(* IEC 61131-3 sources: plc_simulator/services/codesys/POUs (part 4) *)

(* ---- STC_FC_DispatchTask.st ---- *)
(* ===========================================================================================
 *  STC_FC_DispatchTask — Validate and dispatch tasks to transporters
 *
 *  Company : Galvatek part of the John Cockerill Group
 *  Author  : Jarmo Piipponen
 *  Created : 25.03.2026
 *
 * -------------------------------------------------------------------------------------------
 *  Called every PLC scan from MainScheduler.
 *  For each idle transporter with queued tasks:
 *  1. Skip if transporter not idle or queue empty
 *  2. Time check: start_time close enough?
 *  3. Sink station free check (with parallel alternatives)
 *  4. Conflict check against active transporters
 *  5. Dispatch: write to TransporterStatus → RunTasks picks it up
 *
 *  ------------------------------------------------------------------------------------------
 *
 *  Changes:
 *
 *
 *
 *)

FUNCTION STC_FC_DispatchTask : BOOL

(* Introduction of Variables ----------------------------------------------------------------*)

VAR_EXTERNAL CONSTANT
    MAX_TRANSPORTERS        : INT;
    MAX_UNITS               : INT;
    MAX_STATIONS_PER_STEP   : INT;
    MAX_STEPS_PER_PROGRAM   : INT;
    MIN_STATION_INDEX        : INT;
    MAX_STATION_INDEX        : INT;
    SCH_DISPATCH_MARGIN_S   : REAL;
    USED                    : INT;
    PROCESSED               : INT;
END_VAR

VAR_EXTERNAL
  TransporterStatus             : ARRAY[1..MAX_TRANSPORTERS] OF UDT_TransporterStatusType;
  Task                    : ARRAY[1..MAX_TRANSPORTERS] OF UDT_JC_TskQueueType;
  Stations                 : ARRAY[MIN_STATION_INDEX..MAX_STATION_INDEX] OF UDT_StationType;
  StationOccupancy             : ARRAY[1..MAX_STATION_INDEX] OF UDT_JC_UnitAtStationType;
  Unit                    : ARRAY[1..MAX_UNITS] OF UDT_JC_UnitType;
  TreatmentPrograms                 : ARRAY[1..MAX_UNITS] OF UDT_TreatmentProgramType;
  Ntt                     : ARRAY[1..MAX_TRANSPORTERS] OF UDT_JC_NttTransporterType;
  Batch                   : ARRAY[1..MAX_UNITS] OF UDT_BatchType;
  Move                    : ARRAY[1..MAX_TRANSPORTERS] OF UDT_JC_MoveTimesType;
  Transporters                     : ARRAY[0..MAX_TRANSPORTERS] OF UDT_TransporterType;
  Schedule                : ARRAY[1..MAX_UNITS] OF UDT_JC_TskScheduleType;
  TimeS                  : LINT;
  EventPending           : UDT_JC_EventMsgType;
  EventPendingValid     : BOOL;
  DispatchedTask         : ARRAY[1..MAX_TRANSPORTERS] OF UDT_JC_DispatchedTaskType;
END_VAR

VAR
  vTi                        : INT;     (* transporter loop *)
  (* Task fields — read from queue[1] to avoid struct copy *)
  vTUnit                    : INT;
  vTStage                   : INT;
  vTLift                    : INT;
  vTSink                    : INT;
  vTStart                   : LINT;
  vTFinish                  : LINT;
  vTCalcTime               : DINT;
  (* Time check *)
  vTravelS                  : REAL;
  vMarginS                  : LINT;
  vFromIdx                  : INT;
  vToIdx                    : INT;
  (* Sink search *)
  vSinkStn                  : INT;
  vSinkFree                 : BOOL;
  vBestStn                  : INT;
  vBestChange               : LINT;
  vSi                        : INT;
  vCandStn                  : INT;
  vCandFree                 : BOOL;
  vUj                        : INT;
  vTgt                       : INT;
  vNttIdx                   : INT;     (* resolved NTT index (buffer 6/7/8) *)
  vNttCnt                   : INT;
  vNttFbCnt                : INT;
  (* Conflict check *)
  vConflict                  : BOOL;
  vCj                        : INT;
  vTaskMin                  : INT;     (* min station of our proposed task *)
  vTaskMax                  : INT;     (* max station of our proposed task *)
  (* Queue position loop *)
  vQi                        : INT;
  (* Shift-down after dispatch *)
  vSh                        : INT;
  (* Transfer time for batch progress bar *)
  vXferTotal                : REAL;
  (* Program stage number for event *)
  vProgStage                : INT;
  (* Manual task dispatch flag *)
  vUnitOk                   : BOOL;
END_VAR

FOR vTi := 1 TO MAX_TRANSPORTERS DO

  (* ── 1. Skip if not idle or queue empty ── *)
  (* Accept idle (Phase=0) OR move-away in progress (Phase=1, Status=3) *)
  IF (TransporterStatus[vTi].Phase = 0 OR (TransporterStatus[vTi].Phase = 1 AND TransporterStatus[vTi].Status = 3))
     AND Task[vTi].Count >= 1 THEN

    (* Try each queue position — skip blocked tasks, dispatch first feasible *)
    FOR vQi := 1 TO Task[vTi].Count DO

    (* Read task fields from queue position vQi *)
    vTUnit      := Task[vTi].Queue[vQi].Unit;
    vTStage     := Task[vTi].Queue[vQi].Stage;  (* schedule index *)
    vTLift      := Task[vTi].Queue[vQi].LiftStationTarget;
    vTSink      := Task[vTi].Queue[vQi].SinkStationTarget;
    vTStart     := Task[vTi].Queue[vQi].StartTime;
    vTFinish    := Task[vTi].Queue[vQi].FinishTime;
    vTCalcTime := Task[vTi].Queue[vQi].CalcTime;

    (* Queue[].Stage already contains ProgramStage (set by STC_FC_CreateTasks) *)
    vProgStage := vTStage;

    (* ── 1b. Lift station unit check — unit must be AT the lift station ── *)
    (* Manual tasks have Unit=0 → skip unit-location check *)
    (* NOTE: CODESYS does NOT short-circuit OR — use nested IFs *)
    vUnitOk := FALSE;
    IF vTUnit = 0 THEN
      vUnitOk := TRUE;
    ELSIF vTUnit >= 1 AND vTUnit <= MAX_UNITS THEN
      IF Unit[vTUnit].location = vTLift THEN
        vUnitOk := TRUE;
      END_IF;
    END_IF;

    IF vUnitOk THEN

    (* ── 2. Time check ── *)
    vTravelS := 0.0;
    IF TransporterStatus[vTi].CurrentStation > 0 AND vTLift > 0
       AND TransporterStatus[vTi].CurrentStation <> vTLift THEN
      vFromIdx := TransporterStatus[vTi].CurrentStation - MIN_STATION_INDEX;
      vToIdx   := vTLift - MIN_STATION_INDEX;
      IF vFromIdx >= 1 AND vFromIdx <= 30 AND vToIdx >= 1 AND vToIdx <= 30 THEN
        vTravelS := INT_TO_REAL(Move[vTi].Travel[vFromIdx].ToTime[vToIdx]) / 10.0;
      END_IF;
    END_IF;

    vMarginS := vTStart - TimeS;

    IF vMarginS <= REAL_TO_LINT(vTravelS + SCH_DISPATCH_MARGIN_S) THEN

      (* ── 3. Sink station free check ── *)
      vSinkStn := vTSink;
      vSinkFree := FALSE;

      IF vSinkStn >= MIN_STATION_INDEX AND vSinkStn <= MAX_STATION_INDEX THEN
        vSinkFree := TRUE;
        FOR vUj := 1 TO MAX_UNITS DO
          IF Unit[vUj].location = vSinkStn AND Unit[vUj].Status = USED THEN
            vSinkFree := FALSE;
          END_IF;
        END_FOR;
      END_IF;

      IF NOT vSinkFree THEN
        (* Search alternative parallel stations *)
        vBestStn := 0;
        vBestChange := LINT#2000000000;

        IF vProgStage >= 1 AND vProgStage <= MAX_STEPS_PER_PROGRAM
           AND vTUnit >= 1 AND vTUnit <= MAX_UNITS THEN
          (* Treatment task — look in TreatmentPrograms for parallel stations *)
          FOR vSi := 0 TO MAX_STATIONS_PER_STEP - 1 DO
            vCandStn := TreatmentPrograms[vTUnit].Steps[vProgStage].Stations[vSi];
            IF vCandStn > 0 AND vCandStn <> vTSink THEN
              IF vCandStn >= MIN_STATION_INDEX AND vCandStn <= MAX_STATION_INDEX THEN
                vCandFree := TRUE;
                FOR vUj := 1 TO MAX_UNITS DO
                  IF Unit[vUj].location = vCandStn AND Unit[vUj].Status = USED THEN
                    vCandFree := FALSE;
                  END_IF;
                END_FOR;
                IF vCandFree THEN
                  IF StationOccupancy[vCandStn].ChangeTime < vBestChange THEN
                    vBestChange := StationOccupancy[vCandStn].ChangeTime;
                    vBestStn := vCandStn;
                  END_IF;
                END_IF;
              END_IF;
            END_IF;
          END_FOR;

        ELSIF vProgStage = 0 AND vTUnit >= 1 AND vTUnit <= MAX_UNITS THEN
          (* No-treatment task — look in Ntt for alternatives *)
          vTgt := Unit[vTUnit].Target;
          IF vTgt >= 1 AND vTgt <= 5 THEN
            (* Resolve buffer NTT index like NoTreatment does *)
            IF vTgt = 2 THEN
              IF Batch[vTUnit].BatchCode = 0 THEN
                vNttIdx := 6;
              ELSIF Batch[vTUnit].State = PROCESSED THEN
                vNttIdx := 8;
              ELSE
                vNttIdx := 7;
              END_IF;
            ELSE
              vNttIdx := vTgt;
            END_IF;
            (* Check primary stations *)
            vNttCnt := Ntt[vTi].Target[vNttIdx].StationCount;
            FOR vSi := 1 TO vNttCnt DO
              IF vSi <= MAX_STATIONS_PER_STEP THEN
                vCandStn := Ntt[vTi].Target[vNttIdx].Stations[vSi];
                IF vCandStn > 0 AND vCandStn <> vTSink THEN
                  IF vCandStn >= MIN_STATION_INDEX AND vCandStn <= MAX_STATION_INDEX THEN
                    vCandFree := TRUE;
                    FOR vUj := 1 TO MAX_UNITS DO
                      IF Unit[vUj].location = vCandStn AND Unit[vUj].Status = USED THEN
                        vCandFree := FALSE;
                      END_IF;
                    END_FOR;
                    IF vCandFree THEN
                      IF StationOccupancy[vCandStn].ChangeTime < vBestChange THEN
                        vBestChange := StationOccupancy[vCandStn].ChangeTime;
                        vBestStn := vCandStn;
                      END_IF;
                    END_IF;
                  END_IF;
                END_IF;
              END_IF;
            END_FOR;
            (* Check fallback stations *)
            vNttFbCnt := Ntt[vTi].Target[vNttIdx].FallbackCount;
            FOR vSi := 1 TO vNttFbCnt DO
              IF vSi <= MAX_STATIONS_PER_STEP THEN
                vCandStn := Ntt[vTi].Target[vNttIdx].FallbackStations[vSi];
                IF vCandStn > 0 AND vCandStn <> vTSink THEN
                  IF vCandStn >= MIN_STATION_INDEX AND vCandStn <= MAX_STATION_INDEX THEN
                    vCandFree := TRUE;
                    FOR vUj := 1 TO MAX_UNITS DO
                      IF Unit[vUj].location = vCandStn AND Unit[vUj].Status = USED THEN
                        vCandFree := FALSE;
                      END_IF;
                    END_FOR;
                    IF vCandFree THEN
                      IF StationOccupancy[vCandStn].ChangeTime < vBestChange THEN
                        vBestChange := StationOccupancy[vCandStn].ChangeTime;
                        vBestStn := vCandStn;
                      END_IF;
                    END_IF;
                  END_IF;
                END_IF;
              END_IF;
            END_FOR;
          END_IF;
        END_IF;

        IF vBestStn > 0 THEN
          vSinkStn := vBestStn;
          vSinkFree := TRUE;
        END_IF;
      END_IF;  (* NOT vSinkFree *)

      IF vSinkFree THEN

        (* ── 4. Conflict check ── *)
        vConflict := FALSE;

        IF vTLift <= vSinkStn THEN
          vTaskMin := vTLift;
          vTaskMax := vSinkStn;
        ELSE
          vTaskMin := vSinkStn;
          vTaskMax := vTLift;
        END_IF;

        FOR vCj := 1 TO MAX_TRANSPORTERS DO
          IF vCj <> vTi AND TransporterStatus[vCj].Phase > 0 THEN

            (* a) T2's entire active task inside our range → vConflict *)
            IF TransporterStatus[vCj].LiftStationTarget >= vTaskMin
               AND TransporterStatus[vCj].LiftStationTarget <= vTaskMax
               AND TransporterStatus[vCj].SinkStationTarget >= vTaskMin
               AND TransporterStatus[vCj].SinkStationTarget <= vTaskMax THEN
              vConflict := TRUE;
            END_IF;

            (* b) T2 delivers to one of our exact stations → vConflict *)
            IF TransporterStatus[vCj].SinkStationTarget = vTLift
               OR TransporterStatus[vCj].SinkStationTarget = vSinkStn THEN
              vConflict := TRUE;
            END_IF;

          END_IF;
        END_FOR;

        IF NOT vConflict THEN
          (* ── 5. Dispatch: assign task to transporter ── *)
          TransporterStatus[vTi].TaskId      := vTStart;
          TransporterStatus[vTi].LiftStationTarget := vTLift;
          TransporterStatus[vTi].SinkStationTarget := vSinkStn;
          TransporterStatus[vTi].CurrentTaskFinishTime := Task[vTi].Queue[vQi].FinishTime;
          StationOccupancy[vTi].UnitId      := vTUnit;
          TransporterStatus[vTi].TaskRemainingTime := vTCalcTime;

          (* ── 5b. Fill dispatched task package ── *)
          DispatchedTask[vTi].TaskId           := vTStart;
          DispatchedTask[vTi].UnitId           := vTUnit;
          DispatchedTask[vTi].LiftStation      := vTLift;
          DispatchedTask[vTi].SinkStation      := vSinkStn;
          IF vTLift >= MIN_STATION_INDEX AND vTLift <= MAX_STATION_INDEX THEN
            DispatchedTask[vTi].LiftX              := Stations[vTLift].XPosition;
            DispatchedTask[vTi].LiftKind           := Stations[vTLift].DryWet;
            DispatchedTask[vTi].DroppingTime_x10   := Stations[vTLift].DrippingTime;
            DispatchedTask[vTi].LiftDeviceDelay_x10 := Stations[vTLift].DeviceDelay;
          END_IF;
          IF vSinkStn >= MIN_STATION_INDEX AND vSinkStn <= MAX_STATION_INDEX THEN
            DispatchedTask[vTi].SinkX              := Stations[vSinkStn].XPosition;
            DispatchedTask[vTi].SinkKind           := Stations[vSinkStn].DryWet;
            DispatchedTask[vTi].SinkDeviceDelay_x10 := Stations[vSinkStn].DeviceDelay;
          END_IF;
          DispatchedTask[vTi].DripTrayDelay_x10 := Transporters[vTi].DripTrayDelay;
          DispatchedTask[vTi].TreatmentTime    := vTCalcTime;
          DispatchedTask[vTi].MinTime          := Task[vTi].Queue[vQi].MinTime;
          DispatchedTask[vTi].MaxTime          := Task[vTi].Queue[vQi].MaxTime;
          DispatchedTask[vTi].NttPrimary       := Task[vTi].Queue[vQi].NttPrimary;
          IF vTUnit >= 1 AND vTUnit <= MAX_UNITS THEN
            DispatchedTask[vTi].BatchCode      := Batch[vTUnit].BatchCode;
            DispatchedTask[vTi].ProgramStage   := Batch[vTUnit].CurStage;
          ELSE
            DispatchedTask[vTi].BatchCode      := 0;
            DispatchedTask[vTi].ProgramStage   := 0;
          END_IF;
          DispatchedTask[vTi].Active           := TRUE;

          (* ── Emit TASK_DISPATCHED event (msg_type=1) ── *)
          vXferTotal := STC_FC_CalcTransferTime(
            iFromStn            := vTLift,
            iToStn              := vSinkStn,
            iMove                := Move[vTi],
            iFromDroppingX10   := Stations[vTLift].DrippingTime,
            iToDeviceDelayX10 := Stations[vSinkStn].DeviceDelay,
            iDripTrayDelayX10 := Transporters[vTi].DripTrayDelay
          );
          IF vXferTotal < 1.0 THEN
            vXferTotal := INT_TO_REAL(ABS(vSinkStn - vTLift)) * 8.0;
          END_IF;
  IF vXferTotal < 5.0 THEN vXferTotal := 60.0; END_IF;
          DispatchedTask[vTi].TransferTime_x10 := REAL_TO_DINT(vXferTotal * 10.0);
          IF NOT EventPendingValid THEN
            EventPending.MsgType := 1;
            EventPending.TsHi := LINT_TO_UINT(TimeS / LINT#65536);
            EventPending.TsLo := LINT_TO_UINT(TimeS MOD LINT#65536);
            EventPending.Payload[1]  := LINT_TO_INT(vTStart / LINT#65536);   (* TaskId_Hi *)
            EventPending.Payload[2]  := LINT_TO_INT(vTStart MOD LINT#65536);  (* TaskId_Lo *)
            EventPending.Payload[3]  := vTi;
            EventPending.Payload[4]  := vTUnit;
            EventPending.Payload[5]  := vTLift;
            EventPending.Payload[6]  := vSinkStn;
            IF vTUnit >= 1 AND vTUnit <= MAX_UNITS THEN
              vProgStage := Batch[vTUnit].CurStage;
              EventPending.Payload[7]  := vProgStage;
              EventPending.Payload[8]  := Batch[vTUnit].BatchCode;
            ELSE
              EventPending.Payload[7]  := 0;
              EventPending.Payload[8]  := 0;
            END_IF;
            EventPending.Payload[9]  := DINT_TO_INT(vTCalcTime);
            EventPending.Payload[10] := DINT_TO_INT(Task[vTi].Queue[vQi].MinTime);
            EventPending.Payload[11] := DINT_TO_INT(Task[vTi].Queue[vQi].MaxTime);
            EventPending.Payload[12] := REAL_TO_INT(vXferTotal);
            EventPendingValid := TRUE;
          END_IF;

          (* Copy station-specific timing from config *)
          IF vTLift >= MIN_STATION_INDEX AND vTLift <= MAX_STATION_INDEX THEN
            TransporterStatus[vTi].DrippingTime := Stations[vTLift].DrippingTime;
          END_IF;

          (* Shift queue: remove position vQi, move rest up *)
          FOR vSh := vQi + 1 TO Task[vTi].Count DO
            Task[vTi].Queue[vSh - 1] := Task[vTi].Queue[vSh];
          END_FOR;
          (* Clear last slot *)
          Task[vTi].Queue[Task[vTi].Count].Unit := 0;
          Task[vTi].Queue[Task[vTi].Count].Stage := 0;
          Task[vTi].Queue[Task[vTi].Count].SrcStage := 0;
          Task[vTi].Queue[Task[vTi].Count].LiftStationTarget := 0;
          Task[vTi].Queue[Task[vTi].Count].SinkStationTarget := 0;
          Task[vTi].Queue[Task[vTi].Count].StartTime := 0;
          Task[vTi].Queue[Task[vTi].Count].FinishTime := 0;
          Task[vTi].Queue[Task[vTi].Count].CalcTime := 0;
          Task[vTi].Queue[Task[vTi].Count].MinTime := 0;
          Task[vTi].Queue[Task[vTi].Count].MaxTime := 0;
          Task[vTi].Count := Task[vTi].Count - 1;
          EXIT;  (* dispatched — stop searching this queue *)

        END_IF;  (* NOT vConflict *)

      END_IF;  (* vSinkFree *)

    END_IF;  (* time check *)

    END_IF;  (* unit at lift station *)

    END_FOR;  (* vQi — try next queue position *)

  END_IF;  (* idle + queue *)

END_FOR;

STC_FC_DispatchTask := TRUE;

END_FUNCTION

(* ---- STC_FC_ManualTask.st ---- *)
(* ===========================================================================================
 *  STC_FC_ManualTask — Execute manual transport tasks from gateway
 *
 *  Company : Galvatek part of the John Cockerill Group
 *  Author  : Jarmo Piipponen
 *  Created : 25.03.2026
 *
 * -------------------------------------------------------------------------------------------
 *  For each transporter, checks ManualTask[vTi].Valid.
 *  If the transporter is idle (Phase=0), validates stations,
 *  calculates transfer time, and inserts a task into the queue
 *  (same pattern as TSK_FC_NoTreatment).
 *  Clears Valid after task is created, or on invalid input.
 *
 *  Called from TSK_FB_Scheduler phase 2200 (before NTT).
 *
 * ------------------------------------------------------------------------------------------
 *
 *  Changes:
 *
 *
 *
 *)

FUNCTION STC_FC_ManualTask : BOOL

(* Introduction of Variables ----------------------------------------------------------------*)

VAR_INPUT
  iTimeS                  : LINT;
END_VAR

VAR_IN_OUT
  ioTask                   : ARRAY[1..MAX_TRANSPORTERS] OF UDT_JC_TskQueueType;
END_VAR

VAR_EXTERNAL
  ManualTask             : ARRAY[1..MAX_TRANSPORTERS] OF UDT_JC_ManualTaskType;
  TransporterStatus             : ARRAY[1..MAX_TRANSPORTERS] OF UDT_TransporterStatusType;
  Move                    : ARRAY[1..MAX_TRANSPORTERS] OF UDT_JC_MoveTimesType;
  Unit                    : ARRAY[1..MAX_UNITS] OF UDT_JC_UnitType;
  Stations                  : ARRAY[MIN_STATION_INDEX..MAX_STATION_INDEX] OF UDT_StationType;
  Transporters              : ARRAY[0..MAX_TRANSPORTERS] OF UDT_TransporterType;
END_VAR

VAR_EXTERNAL CONSTANT
  MAX_TASK_QUEUE            : INT;
  MAX_UNITS                 : INT;
  USED                      : INT;
END_VAR

VAR
  vTi                        : INT;
  vAi                        : INT;
  vSh                        : INT;
  vLift                      : INT;
  vSink                      : INT;
  vCovers                    : BOOL;
  vTransPos                 : INT;
  vTmpMove                  : UDT_JC_MoveTimesType;
  vXferS                    : REAL;
  vTravelToLiftS          : REAL;
  vTaskStart                : LINT;
  vTaskEnd                  : LINT;
END_VAR

STC_FC_ManualTask := TRUE;

FOR vTi := 1 TO MAX_TRANSPORTERS DO
  IF NOT ManualTask[vTi].Valid THEN
    CONTINUE;
  END_IF;

  vLift := ManualTask[vTi].LiftStation;
  vSink := ManualTask[vTi].SinkStation;

  (* Validate station range *)
  IF vLift < MIN_STATION_INDEX OR vLift > MAX_STATION_INDEX
     OR vSink < MIN_STATION_INDEX OR vSink > MAX_STATION_INDEX
     OR vLift = vSink THEN
    ManualTask[vTi].Valid := FALSE;
    CONTINUE;
  END_IF;

  (* Transporter must be active and idle *)
  (* Transporter must be active and idle or in move-away *)
  IF NOT TransporterStatus[vTi].IsActive THEN
    CONTINUE;
  END_IF;
  IF TransporterStatus[vTi].Phase <> 0
     AND NOT (TransporterStatus[vTi].Phase = 1 AND TransporterStatus[vTi].Status = 3) THEN
    CONTINUE;  (* keep Valid — retry next cycle *)
  END_IF;

  (* Check vLift station is within transporter TaskArea *)
  vCovers := FALSE;
  FOR vAi := 1 TO 4 DO
    IF Transporters[vTi].TaskArea[vAi].MinLift > 0
       OR Transporters[vTi].TaskArea[vAi].MaxLift > 0 THEN
      IF vLift >= Transporters[vTi].TaskArea[vAi].MinLift
         AND vLift <= Transporters[vTi].TaskArea[vAi].MaxLift THEN
        vCovers := TRUE;
      END_IF;
    END_IF;
  END_FOR;

  IF NOT vCovers THEN
    ManualTask[vTi].Valid := FALSE;
    CONTINUE;
  END_IF;

  (* Calculate transfer time *)
  vTmpMove := Move[vTi];
  vXferS := STC_FC_CalcTransferTime(
    iFromStn            := vLift,
    iToStn              := vSink,
    iMove                := vTmpMove,
    iFromDroppingX10   := Stations[vLift].DrippingTime,
    iToDeviceDelayX10 := Stations[vSink].DeviceDelay,
    iDripTrayDelayX10 := Transporters[vTi].DripTrayDelay);

  (* Calculate travel-to-vLift: time for transporter to reach vLift station *)
  vTravelToLiftS := 0.0;
  vTransPos := TransporterStatus[vTi].CurrentStation;
  IF vTransPos > 0 AND vTransPos <> vLift THEN
    vTravelToLiftS := STC_FC_CalcHorizontalTravel(
      iFromStn := vTransPos,
      iToStn   := vLift,
      iMove     := vTmpMove);
  END_IF;

  vTaskStart := iTimeS + REAL_TO_LINT(vTravelToLiftS);
  vTaskEnd   := vTaskStart + REAL_TO_LINT(vXferS);

  (* Check vSink station is free — no unit occupying it *)
  vCovers := TRUE;  (* reuse variable as sink_free flag *)
  FOR vSh := 1 TO MAX_UNITS DO
    IF Unit[vSh].location = vSink AND Unit[vSh].Status = USED THEN
      vCovers := FALSE;
    END_IF;
  END_FOR;
  IF NOT vCovers THEN
    ManualTask[vTi].Valid := FALSE;
    CONTINUE;
  END_IF;

  (* Insert task at queue position 1 *)
  IF ioTask[vTi].Count < MAX_TASK_QUEUE THEN
    FOR vSh := ioTask[vTi].Count TO 1 BY -1 DO
      ioTask[vTi].Queue[vSh + 1] := ioTask[vTi].Queue[vSh];
    END_FOR;
    ioTask[vTi].Queue[1].Unit              := 0;
    ioTask[vTi].Queue[1].Stage             := 0;
    ioTask[vTi].Queue[1].LiftStationTarget := vLift;
    ioTask[vTi].Queue[1].SinkStationTarget := vSink;
    ioTask[vTi].Queue[1].StartTime         := vTaskStart;
    ioTask[vTi].Queue[1].FinishTime        := vTaskEnd;
    ioTask[vTi].Queue[1].CalcTime          := 0;
    ioTask[vTi].Queue[1].MinTime           := 0;
    ioTask[vTi].Queue[1].MaxTime           := 0;
    ioTask[vTi].Queue[1].NttPrimary        := 0;
    ioTask[vTi].Count := ioTask[vTi].Count + 1;
  END_IF;

  ManualTask[vTi].Valid := FALSE;
END_FOR;

END_FUNCTION

(* ---- STC_FC_NoTreatmentStates.st ---- *)
(* ===========================================================================================
 *  STC_FC_NoTreatmentStates — Non-treatment target state management
 *
 *  Company : Galvatek part of the John Cockerill Group
 *  Author  : Jarmo Piipponen
 *  Created : 25.03.2026
 *
 * -------------------------------------------------------------------------------------------
 *  Manages non-treatment target states for all units.
 *
 *  Structure:
 *  Pass 0 — SNAPSHOT: read unit/batch/station state into vSnap[]
 *  Section 1 — PROCESSED: mark last-stage units as PROCESSED
 *  Section 2 — TO_AVOID: clear occupied next-stage stations
 *  Section 3 — TO_LOADING: route one empty unit to loading
 *
 *  ------------------------------------------------------------------------------------------
 *
 *  Changes:
 *
 *
 *
 *)

FUNCTION STC_FC_NoTreatmentStates : BOOL

(* Introduction of Variables ----------------------------------------------------------------*)

VAR_EXTERNAL CONSTANT
    MAX_UNITS               : INT;
    MAX_STEPS_PER_PROGRAM   : INT;
    MAX_STATIONS_PER_STEP   : INT;
    MIN_STATION_INDEX        : INT;
    MAX_STATION_INDEX        : INT;
    IN_PROCESS              : INT;
    PROCESSED               : INT;
    NOT_USED                : INT;
    TO_NONE                 : INT;
    TO_UNLOAD               : INT;
    TO_AVOID                : INT;
    TO_LOADING              : INT;
    USED                    : INT;
    OP_BUFFER               : INT;
    OP_BUFFER_PROCESSED     : INT;
    OP_LOADING              : INT;
    OP_LOADING_UNLOADING    : INT;
END_VAR

VAR_EXTERNAL
  Unit                    : ARRAY[1..MAX_UNITS] OF UDT_JC_UnitType;
  Batch                   : ARRAY[1..MAX_UNITS] OF UDT_BatchType;
  TreatmentPrograms                 : ARRAY[1..MAX_UNITS] OF UDT_TreatmentProgramType;
  Stations                 : ARRAY[MIN_STATION_INDEX..MAX_STATION_INDEX] OF UDT_StationType;
  StationOccupancy             : ARRAY[1..MAX_STATION_INDEX] OF UDT_JC_UnitAtStationType;
  TimeS                  : LINT;
  ProductionQueue        : INT;
  EventPending           : UDT_JC_EventMsgType;
  EventPendingValid     : BOOL;
END_VAR

VAR
  (* Snapshot *)
  vSnap                      : ARRAY[1..MAX_UNITS] OF UDT_JC_UnitSnapType;
  vU                         : INT;        (* unit loop index *)
  vHasLoading               : BOOL;       (* any unit already has TO_LOADING *)
  (* Section 1+2 *)
  vP                         : INT;        (* parallel station loop *)
  vNextStn                  : INT;        (* next stage station *)
  vOccUid                   : INT;        (* unit_id at an occupied station *)
  vFreeFound                : BOOL;       (* any next-stage station is free *)
  vAvoidUid                 : INT;        (* unit to mark TO_AVOID *)
  (* Section 3 *)
  vLoadFree                 : BOOL;       (* a loading station is free *)
  vLoadUid                  : INT;        (* best candidate for TO_LOADING *)
  vLoadInBuf               : BOOL;       (* current candidate is in buffer *)
  vStk                       : INT;        (* station loop *)
  vOp                        : INT;        (* station operation code *)
END_VAR

  (* ════════════════════════════════════════════════════════════
     Pass 0 — SNAPSHOT: collect per-unit state in one pass
     ════════════════════════════════════════════════════════════ *)
  vHasLoading := FALSE;

  FOR vU := 1 TO MAX_UNITS DO
    vSnap[vU].IsActive := Unit[vU].Status <> NOT_USED;
    IF NOT vSnap[vU].IsActive THEN
      CONTINUE;
    END_IF;

    vSnap[vU].Location       := Unit[vU].location;
    vSnap[vU].Target       := Unit[vU].Target;
    vSnap[vU].HasBatch := Batch[vU].BatchCode <> 0;
    vSnap[vU].BatchState    := Batch[vU].State;
    vSnap[vU].CurStage := Batch[vU].CurStage;

    vSnap[vU].OnStation := vSnap[vU].Location >= MIN_STATION_INDEX
                          AND vSnap[vU].Location <= MAX_STATION_INDEX;
    IF vSnap[vU].OnStation THEN
      vSnap[vU].LocationOp    := Stations[vSnap[vU].Location].StationType;
      vSnap[vU].InBuffer := vSnap[vU].LocationOp >= OP_BUFFER AND vSnap[vU].LocationOp <= OP_BUFFER_PROCESSED;
      IF StationOccupancy[vSnap[vU].Location].ChangeTime > 0 THEN
        vSnap[vU].Elapsed := TimeS - StationOccupancy[vSnap[vU].Location].ChangeTime;
      ELSE
        vSnap[vU].Elapsed := 0;
      END_IF;
      IF vSnap[vU].CurStage >= 1 THEN
        vSnap[vU].CalTime := TreatmentPrograms[vU].Steps[vSnap[vU].CurStage].CalTime;
      ELSE
        vSnap[vU].CalTime := 0;
      END_IF;
    ELSE
      vSnap[vU].LocationOp    := 0;
      vSnap[vU].InBuffer := FALSE;
      vSnap[vU].Elapsed   := 0;
      vSnap[vU].CalTime       := 0;
    END_IF;

    IF vSnap[vU].Target = TO_LOADING THEN
      vHasLoading := TRUE;
    END_IF;
  END_FOR;

  (* ════════════════════════════════════════════════════════════
     Section 1 — PROCESSED: mark batch done at last treatment stage
     ════════════════════════════════════════════════════════════ *)
  FOR vU := 1 TO MAX_UNITS DO
    IF NOT vSnap[vU].IsActive OR NOT vSnap[vU].HasBatch THEN
      CONTINUE;
    END_IF;
    IF vSnap[vU].BatchState <> IN_PROCESS OR NOT vSnap[vU].OnStation THEN
      CONTINUE;
    END_IF;
    IF vSnap[vU].CurStage >= 1 AND vSnap[vU].CurStage < MAX_STEPS_PER_PROGRAM THEN
      IF vSnap[vU].CurStage >= TreatmentPrograms[vU].StepCount THEN
        IF vSnap[vU].Elapsed > 0 AND vSnap[vU].Elapsed >= DINT_TO_LINT(vSnap[vU].CalTime) THEN
          Batch[vU].State := PROCESSED;
          vSnap[vU].BatchState   := PROCESSED;  (* update snapshot *)

          (* ── Emit BATCH_COMPLETED event (msg_type=5) ── *)
          IF NOT EventPendingValid THEN
            EventPending.MsgType := 5;
            EventPending.TsHi := LINT_TO_UINT(TimeS / LINT#65536);
            EventPending.TsLo := LINT_TO_UINT(TimeS MOD LINT#65536);
            EventPending.Payload[1]  := vU;                                  (* unit_id *)
            EventPending.Payload[2]  := Batch[vU].BatchCode;               (* batch_code *)
            EventPending.Payload[3]  := TreatmentPrograms[vU].StepCount;             (* stage_count *)
            EventPending.Payload[4]  := vSnap[vU].Location;                   (* final_station *)
            EventPending.Payload[5]  := 0;
            EventPending.Payload[6]  := 0;
            EventPending.Payload[7]  := 0;
            EventPending.Payload[8]  := 0;
            EventPending.Payload[9]  := 0;
            EventPending.Payload[10] := 0;
            EventPending.Payload[11] := 0;
            EventPending.Payload[12] := 0;
            EventPendingValid := TRUE;
          END_IF;

          (* Route to unloading station *)
          IF vSnap[vU].Target = TO_NONE THEN
            Unit[vU].Target := TO_UNLOAD;
            vSnap[vU].Target   := TO_UNLOAD;
          END_IF;
        END_IF;
      END_IF;
    END_IF;
  END_FOR;

  (* ════════════════════════════════════════════════════════════
     Section 2 — TO_AVOID: clear the way to next treatment station
     ════════════════════════════════════════════════════════════ *)
  FOR vU := 1 TO MAX_UNITS DO
    IF NOT vSnap[vU].IsActive OR NOT vSnap[vU].HasBatch THEN
      CONTINUE;
    END_IF;
    IF vSnap[vU].BatchState <> IN_PROCESS THEN
      CONTINUE;
    END_IF;
    IF vSnap[vU].CurStage < 1 OR vSnap[vU].CurStage >= MAX_STEPS_PER_PROGRAM THEN
      CONTINUE;
    END_IF;
    IF vSnap[vU].CurStage >= TreatmentPrograms[vU].StepCount THEN
      CONTINUE;  (* no next stage *)
    END_IF;

    (* — Pass 1: any next-stage station free or being cleared? — *)
    vFreeFound := FALSE;
    vAvoidUid  := 0;
    FOR vP := 0 TO MAX_STATIONS_PER_STEP - 1 DO
      vNextStn := TreatmentPrograms[vU].Steps[vSnap[vU].CurStage + 1].Stations[vP];
      IF vNextStn = 0 THEN
        EXIT;
      END_IF;
      IF vNextStn >= MIN_STATION_INDEX AND vNextStn <= MAX_STATION_INDEX THEN
        IF StationOccupancy[vNextStn].UnitId = 0 THEN
          vFreeFound := TRUE;
          EXIT;
        END_IF;
        vOccUid := StationOccupancy[vNextStn].UnitId;
        IF vOccUid >= 1 AND vOccUid <= MAX_UNITS THEN
          IF vSnap[vOccUid].Target = TO_AVOID THEN
            vFreeFound := TRUE;
            EXIT;
          END_IF;
        END_IF;
      END_IF;
    END_FOR;

    (* — Pass 2: all occupied → mark ONE movable unit TO_AVOID — *)
    IF NOT vFreeFound THEN
      FOR vP := 0 TO MAX_STATIONS_PER_STEP - 1 DO
        vNextStn := TreatmentPrograms[vU].Steps[vSnap[vU].CurStage + 1].Stations[vP];
        IF vNextStn = 0 THEN
          EXIT;
        END_IF;
        IF vNextStn >= MIN_STATION_INDEX AND vNextStn <= MAX_STATION_INDEX THEN
          vOccUid := StationOccupancy[vNextStn].UnitId;
          IF vOccUid >= 1 AND vOccUid <= MAX_UNITS THEN
            IF NOT vSnap[vOccUid].HasBatch AND vSnap[vOccUid].Target = TO_NONE THEN
              vAvoidUid := vOccUid;
              EXIT;
            END_IF;
          END_IF;
        END_IF;
      END_FOR;

      IF vAvoidUid >= 1 THEN
        Unit[vAvoidUid].Target := TO_AVOID;
        vSnap[vAvoidUid].Target     := TO_AVOID;  (* update snapshot *)
      END_IF;
    END_IF;
  END_FOR;

  (* ════════════════════════════════════════════════════════════
     Section 3 — TO_LOADING: route one empty unit to loading station
     ════════════════════════════════════════════════════════════ *)
  IF ProductionQueue = 1 AND NOT vHasLoading THEN

    (* Check if any loading station is free *)
    vLoadFree := FALSE;
    FOR vStk := MIN_STATION_INDEX TO MAX_STATION_INDEX DO
      vOp := Stations[vStk].StationType;
      IF (vOp = OP_LOADING OR vOp = OP_LOADING_UNLOADING)
         AND StationOccupancy[vStk].UnitId = 0 THEN
        vLoadFree := TRUE;
        EXIT;
      END_IF;
    END_FOR;

    IF vLoadFree THEN
      vLoadUid    := 0;
      vLoadInBuf := FALSE;
      FOR vU := 1 TO MAX_UNITS DO
        IF vSnap[vU].IsActive AND NOT vSnap[vU].HasBatch
           AND vSnap[vU].Target = TO_NONE AND vSnap[vU].OnStation THEN
          IF vSnap[vU].InBuffer THEN
            IF vLoadUid = 0 THEN
              vLoadUid    := vU;
              vLoadInBuf := TRUE;
            END_IF;
          ELSE
            IF vLoadUid = 0 OR vLoadInBuf THEN
              vLoadUid    := vU;
              vLoadInBuf := FALSE;
            END_IF;
          END_IF;
        END_IF;
      END_FOR;

      IF vLoadUid >= 1 THEN
        Unit[vLoadUid].Target := TO_LOADING;
      END_IF;
    END_IF; (* vLoadFree *)

  END_IF; (* production_queue AND NOT vHasLoading *)

  STC_FC_NoTreatmentStates := TRUE;

END_FUNCTION

(* ---- STC_FC_ShiftSchedule.st ---- *)
(* ===========================================================================================
 *  STC_FC_ShiftSchedule — Shift schedule + task times
 *
 *  Company : Galvatek part of the John Cockerill Group
 *  Author  : Jarmo Piipponen
 *  Created : 25.03.2026
 *
 * -------------------------------------------------------------------------------------------
 *  Propagates a time shift through one unit's schedule stages
 *  AND through all matching tasks.
 *
 *  Positive iAmount = DELAY (shift later),
 *  Negative iAmount = ADVANCE (shift earlier).
 *
 *  VAR_IN_OUT: ioSchedule, ioTask — caller passes live or
 *  workspace arrays.
 *
 *  ------------------------------------------------------------------------------------------
 *
 *  Changes:
 *
 *
 *
 *)

FUNCTION STC_FC_ShiftSchedule : BOOL

(* Introduction of Variables ----------------------------------------------------------------*)

VAR_INPUT
  iUnit                    : INT;     (* unit index 1..10 *)
  iFromStage              : INT;     (* propagate from this stage onward *)
  iAmount                  : REAL;    (* seconds to shift (+ = later, - = earlier) *)
END_VAR

VAR_IN_OUT  (* array sizes must match GVL_JC_Constants: 10=MAX_UNITS, 3=MAX_TRANSPORTERS *)
  ioSchedule               : ARRAY[1..10] OF UDT_JC_TskScheduleType;
  ioTask                   : ARRAY[1..3] OF UDT_JC_TskQueueType;
END_VAR

VAR_EXTERNAL CONSTANT
    MAX_TRANSPORTERS        : INT;
    MAX_UNITS               : INT;
END_VAR

VAR_EXTERNAL
  TimeS                  : LINT;
END_VAR

VAR
  vSc                        : INT;
  vSi                        : INT;
  vQi                        : INT;
  vTi                        : INT;
  vDuration                  : LINT;
END_VAR

STC_FC_ShiftSchedule := TRUE;
IF iUnit < 1 OR iUnit > MAX_UNITS THEN RETURN; END_IF;
IF ABS(iAmount) < 0.001 THEN RETURN; END_IF;

(* -- Shift schedule stages entry/exit times -- *)
vSc := ioSchedule[iUnit].StageCount;
FOR vSi := 1 TO vSc DO
  IF vSi >= 1 AND vSi <= 30
     AND ioSchedule[iUnit].Stages[vSi].ProgramStage >= iFromStage THEN
    ioSchedule[iUnit].Stages[vSi].EntryTime :=
      ioSchedule[iUnit].Stages[vSi].EntryTime + REAL_TO_LINT(iAmount);
    ioSchedule[iUnit].Stages[vSi].ExitTime :=
      ioSchedule[iUnit].Stages[vSi].ExitTime + REAL_TO_LINT(iAmount);
    (* GAP-3: Past-clamp -- don't let EntryTime go before now+1 *)
    IF iAmount < 0.0 AND ioSchedule[iUnit].Stages[vSi].EntryTime < TimeS + LINT#1 THEN
      ioSchedule[iUnit].Stages[vSi].ExitTime := TimeS + LINT#1
        + (ioSchedule[iUnit].Stages[vSi].ExitTime - ioSchedule[iUnit].Stages[vSi].EntryTime);
      ioSchedule[iUnit].Stages[vSi].EntryTime := TimeS + LINT#1;
    END_IF;
  END_IF;
END_FOR;

(* -- Shift matching tasks in all transporter queues -- *)
FOR vTi := 1 TO MAX_TRANSPORTERS DO
  FOR vQi := 1 TO ioTask[vTi].Count DO
    IF ioTask[vTi].Queue[vQi].Unit = iUnit
       AND ioTask[vTi].Queue[vQi].Stage >= iFromStage THEN
      ioTask[vTi].Queue[vQi].StartTime :=
        ioTask[vTi].Queue[vQi].StartTime + REAL_TO_LINT(iAmount);
      ioTask[vTi].Queue[vQi].FinishTime :=
        ioTask[vTi].Queue[vQi].FinishTime + REAL_TO_LINT(iAmount);
      (* GAP-3: Past-clamp -- don't let StartTime go before now+1 *)
      IF iAmount < 0.0 AND ioTask[vTi].Queue[vQi].StartTime < TimeS + LINT#1 THEN
        vDuration := ioTask[vTi].Queue[vQi].FinishTime - ioTask[vTi].Queue[vQi].StartTime;
        ioTask[vTi].Queue[vQi].StartTime := TimeS + LINT#1;
        ioTask[vTi].Queue[vQi].FinishTime := TimeS + LINT#1 + vDuration;
      END_IF;
    END_IF;
  END_FOR;
END_FOR;

END_FUNCTION

(* ---- STC_FC_SortTasks.st ---- *)
(* ===========================================================================================
 *  STC_FC_SortTasks — Insertion sort task queues by priority
 *
 *  Company : Galvatek part of the John Cockerill Group
 *  Author  : Jarmo Piipponen
 *  Created : 25.03.2026
 *
 * -------------------------------------------------------------------------------------------
 *  Shared FC: both TSK and DEP call this with different arrays.
 *  Priority: emergency (overtime ratio > 1.0) first, then
 *  earliest StartTime.
 *
 *  ------------------------------------------------------------------------------------------
 *
 *  Changes:
 *
 *
 *
 *)

FUNCTION STC_FC_SortTasks : BOOL

(* Introduction of Variables ----------------------------------------------------------------*)

VAR_INPUT
  iTrans                   : INT;    (* 0 = all, 1..3 = specific transporter *)
  iTimeS                  : LINT;
END_VAR

VAR_IN_OUT  (* array sizes must match GVL_JC_Constants: 3=MAX_TRANSPORTERS, 10=MAX_UNITS *)
  ioTask                   : ARRAY[1..3] OF UDT_JC_TskQueueType;
  ioBatch                  : ARRAY[1..10] OF UDT_BatchType;
END_VAR

VAR_EXTERNAL CONSTANT
    MAX_TRANSPORTERS        : INT;
    MAX_UNITS               : INT;
    IN_PROCESS              : INT;
END_VAR

VAR_EXTERNAL
  Unit                    : ARRAY[1..MAX_UNITS] OF UDT_JC_UnitType;
END_VAR

VAR
  vTi                        : INT;
  vTStart                   : INT;
  vTEnd                     : INT;
  vInsI                     : INT;
  vInsJ                     : INT;
  vInsCnt                   : INT;
  vTmpTask                  : UDT_JC_TskTaskType;
  vTmpUnit                  : INT;
  vCurUnit                  : INT;
  vTmpRatio                 : REAL;
  vCurRatio                 : REAL;
  vTmpEmerg                 : BOOL;
  vCurEmerg                 : BOOL;
  vDoShift                  : BOOL;
END_VAR

STC_FC_SortTasks := TRUE;

IF iTrans >= 1 AND iTrans <= 3 THEN
  vTStart := iTrans;
  vTEnd   := iTrans;
ELSE
  vTStart := 1;
  vTEnd   := 3;
END_IF;

FOR vTi := vTStart TO vTEnd DO
  vInsCnt := ioTask[vTi].Count;
  IF vInsCnt >= 2 THEN
    FOR vInsI := 2 TO vInsCnt DO
      vTmpTask := ioTask[vTi].Queue[vInsI];

      vTmpRatio := 0.0;
      vTmpUnit  := vTmpTask.Unit;
      IF vTmpUnit >= 1 AND vTmpUnit <= MAX_UNITS THEN
        IF ioBatch[vTmpUnit].State = IN_PROCESS
           AND vTmpTask.Stage >= 1 THEN
          IF ioBatch[vTmpUnit].CurStage = vTmpTask.Stage
             AND Unit[vTmpUnit].location = vTmpTask.LiftStationTarget
             AND ioBatch[vTmpUnit].StartTime > LINT#0
             AND ioBatch[vTmpUnit].MaxTime > 0 THEN
            vTmpRatio := LINT_TO_REAL(iTimeS - ioBatch[vTmpUnit].StartTime)
                         / DINT_TO_REAL(ioBatch[vTmpUnit].MaxTime);
          END_IF;
        END_IF;
      END_IF;
      vTmpEmerg := vTmpRatio > 1.0;

      vInsJ := 0;
      FOR vInsJ := vInsI - 1 TO 1 BY -1 DO
        vCurRatio := 0.0;
        vCurUnit  := ioTask[vTi].Queue[vInsJ].Unit;
        IF vCurUnit >= 1 AND vCurUnit <= MAX_UNITS THEN
          IF ioBatch[vCurUnit].State = IN_PROCESS
             AND ioTask[vTi].Queue[vInsJ].Stage >= 1 THEN
            IF ioBatch[vCurUnit].CurStage = ioTask[vTi].Queue[vInsJ].Stage
               AND Unit[vCurUnit].location = ioTask[vTi].Queue[vInsJ].LiftStationTarget
               AND ioBatch[vCurUnit].StartTime > LINT#0
               AND ioBatch[vCurUnit].MaxTime > 0 THEN
              vCurRatio := LINT_TO_REAL(iTimeS - ioBatch[vCurUnit].StartTime)
                           / DINT_TO_REAL(ioBatch[vCurUnit].MaxTime);
            END_IF;
          END_IF;
        END_IF;
        vCurEmerg := vCurRatio > 1.0;

        vDoShift := FALSE;
        IF vTmpEmerg AND NOT vCurEmerg THEN
          vDoShift := TRUE;
        ELSIF vTmpEmerg AND vCurEmerg THEN
          IF vTmpRatio > vCurRatio THEN
            vDoShift := TRUE;
          END_IF;
        ELSIF NOT vTmpEmerg AND NOT vCurEmerg THEN
          IF ioTask[vTi].Queue[vInsJ].StartTime > vTmpTask.StartTime THEN
            vDoShift := TRUE;
          END_IF;
        END_IF;

        IF NOT vDoShift THEN EXIT; END_IF;

        ioTask[vTi].Queue[vInsJ + 1] := ioTask[vTi].Queue[vInsJ];
      END_FOR;

      ioTask[vTi].Queue[vInsJ + 1] := vTmpTask;
    END_FOR;
  END_IF;
END_FOR;

END_FUNCTION

(* ---- STC_FC_SwapTasks.st ---- *)
(* ===========================================================================================
 *  STC_FC_SwapTasks — Swap same-station task pairs
 *
 *  Company : Galvatek part of the John Cockerill Group
 *  Author  : Jarmo Piipponen
 *  Created : 25.03.2026
 *
 * -------------------------------------------------------------------------------------------
 *  Shared FC: both TSK and DEP call this with different arrays.
 *  Swaps adjacent tasks on the same transporter when the first
 *  task's sink equals the second task's lift (chain optimization).
 *  Returns swap count.
 *
 *  ------------------------------------------------------------------------------------------
 *
 *  Changes:
 *
 *
 *
 *)

FUNCTION STC_FC_SwapTasks : INT   (* returns swap count *)

(* Introduction of Variables ----------------------------------------------------------------*)

VAR_IN_OUT  (* array sizes must match GVL_JC_Constants: 3=MAX_TRANSPORTERS *)
  ioTask                   : ARRAY[1..3] OF UDT_JC_TskQueueType;
END_VAR

VAR_EXTERNAL CONSTANT
    MAX_TRANSPORTERS        : INT;
END_VAR

VAR
  vTi                        : INT;
  vQi                        : INT;
  vCnt                       : INT;
  vTmp                       : UDT_JC_TskTaskType;
  vSwaps                     : INT;
END_VAR

vSwaps := 0;

FOR vTi := 1 TO MAX_TRANSPORTERS DO
  vCnt := ioTask[vTi].Count;
  IF vCnt >= 2 THEN
    FOR vQi := 1 TO vCnt - 1 DO
      IF ioTask[vTi].Queue[vQi].Unit <> ioTask[vTi].Queue[vQi + 1].Unit
         AND ioTask[vTi].Queue[vQi].SinkStationTarget = ioTask[vTi].Queue[vQi + 1].LiftStationTarget THEN
        vTmp := ioTask[vTi].Queue[vQi];
        ioTask[vTi].Queue[vQi] := ioTask[vTi].Queue[vQi + 1];
        ioTask[vTi].Queue[vQi + 1] := vTmp;
        vSwaps := vSwaps + 1;
      END_IF;
    END_FOR;
  END_IF;
END_FOR;

STC_FC_SwapTasks := vSwaps;

END_FUNCTION

(* ---- STC_FC_TakeOut.st ---- *)
(* STC_FC_TakeOut - Evaluate and trigger idle take-out for transporters
   Uses station-specific TakeOutDelay (seconds) and TakeOutDistance (mm) *)
(* IMPORT_MARKER_2026_04_01_B *)

FUNCTION STC_FC_TakeOut : BOOL

VAR_INPUT
  iTimeS                  : LINT;
END_VAR

VAR
  vTi                        : INT;
  vCurrentStation           : INT;
  vTakeOutDelay            : INT;
  vTakeOutDist             : DINT;
  vIdleTime                 : LINT;
  vCurrentX                 : DINT;
  vTargetX                  : DINT;
  vNextLiftX               : DINT;
  vAreaCenter               : DINT;
  vDir                       : INT;
  vQueuedLiftStation       : INT;
  vTimeToStart             : LINT;
  vSi                        : INT;
  vStnX                     : DINT;
  vBestStn                  : INT;
  vBestDist                 : DINT;
  vDx                        : DINT;
END_VAR

STC_FC_TakeOut := TRUE;

FOR vTi := 1 TO MAX_TRANSPORTERS DO

  IF TransporterStatus[vTi].Phase <> 0 THEN CONTINUE; END_IF;
  IF TransporterStatus[vTi].Status <> 3 THEN CONTINUE; END_IF;
  IF NOT TransporterStatus[vTi].IsActive THEN CONTINUE; END_IF;

  vCurrentStation := TransporterStatus[vTi].CurrentStation;
  IF vCurrentStation < MIN_STATION_INDEX OR vCurrentStation > MAX_STATION_INDEX THEN CONTINUE; END_IF;

  vTakeOutDelay := Stations[vCurrentStation].TakeOutDelay;
  IF vTakeOutDelay = 0 THEN CONTINUE; END_IF;

  vTakeOutDist := INT_TO_DINT(Stations[vCurrentStation].TakeOutDistance);
  IF vTakeOutDist <= 0 THEN CONTINUE; END_IF;

  vIdleTime := iTimeS - TransporterStatus[vTi].IdleStartTime;
  IF vIdleTime < DINT_TO_LINT(INT_TO_DINT(vTakeOutDelay)) THEN CONTINUE; END_IF;

  (* Defer if next task on SAME station starts soon *)
  IF Task[vTi].Count > 0 THEN
    vQueuedLiftStation := Task[vTi].Queue[1].LiftStationTarget;
    IF vQueuedLiftStation = vCurrentStation THEN
      vTimeToStart := Task[vTi].Queue[1].StartTime - iTimeS;
      IF vTimeToStart >= 0 AND vTimeToStart < DINT_TO_LINT(INT_TO_DINT(TAKE_OUT_MIN_WAIT_S)) THEN
        CONTINUE;
      END_IF;
    END_IF;
  END_IF;

  vCurrentX := TransporterStatus[vTi].XPosition;

  (* Determine direction: toward next task or toward area center *)
  IF Task[vTi].Count > 0 THEN
    vNextLiftX := Stations[Task[vTi].Queue[1].LiftStationTarget].XPosition;
    IF vNextLiftX > vCurrentX THEN
      vDir := 1;
    ELSE
      vDir := -1;
    END_IF;
  ELSE
    vAreaCenter := (Transporters[vTi].DrivePosMin + Transporters[vTi].DrivePosMax) / 2;
    IF vAreaCenter > vCurrentX THEN
      vDir := 1;
    ELSE
      vDir := -1;
    END_IF;
  END_IF;

  (* Compute minimum target position from TakeOutDistance *)
  vTargetX := vCurrentX + (INT_TO_DINT(vDir) * vTakeOutDist);

  (* Find nearest station in move direction that is at least vTakeOutDist away *)
  vBestStn := 0;
  vBestDist := DINT#2147483647;
  FOR vSi := MIN_STATION_INDEX TO MIN_STATION_INDEX + CountStations - 1 DO
    vStnX := Stations[vSi].XPosition;
    IF vStnX = 0 THEN CONTINUE; END_IF;
    (* Station must be in the correct direction and at least vTakeOutDist from current *)
    IF vDir > 0 THEN
      vDx := vStnX - vCurrentX;
    ELSE
      vDx := vCurrentX - vStnX;
    END_IF;
    IF vDx >= vTakeOutDist AND vDx < vBestDist THEN
      (* Must be within transporter drive limits *)
      IF vStnX >= Transporters[vTi].DrivePosMin AND vStnX <= Transporters[vTi].DrivePosMax THEN
        vBestDist := vDx;
        vBestStn := vSi;
      END_IF;
    END_IF;
  END_FOR;

  IF vBestStn > 0 THEN
    vTargetX := Stations[vBestStn].XPosition;
  ELSE
    CONTINUE;  (* no station found in direction — skip take-out *)
  END_IF;

  (* Skip if we can't actually move *)
  IF ABS(vTargetX - vCurrentX) < 100 THEN CONTINUE; END_IF;

  (* If next task starts soon and take-out would pass over its lift station,
     stop at the lift station instead *)
  IF Task[vTi].Count > 0 THEN
    vTimeToStart := Task[vTi].Queue[1].StartTime - iTimeS;
    IF vTimeToStart >= 0 AND vTimeToStart < DINT_TO_LINT(INT_TO_DINT(TAKE_OUT_MIN_WAIT_S)) THEN
      vQueuedLiftStation := Task[vTi].Queue[1].LiftStationTarget;
      IF vQueuedLiftStation >= MIN_STATION_INDEX AND vQueuedLiftStation <= MAX_STATION_INDEX THEN
        vNextLiftX := Stations[vQueuedLiftStation].XPosition;
        (* Check if take-out target is on the other side of lift station *)
        IF vDir > 0 AND vTargetX > vNextLiftX AND vNextLiftX > vCurrentX THEN
          vTargetX := vNextLiftX;
        ELSIF vDir < 0 AND vTargetX < vNextLiftX AND vNextLiftX < vCurrentX THEN
          vTargetX := vNextLiftX;
        END_IF;
      END_IF;
    END_IF;
  END_IF;

  (* Re-check: still worth moving? *)
  IF ABS(vTargetX - vCurrentX) < 100 THEN CONTINUE; END_IF;

  TransporterStatus[vTi].Phase := 1;
  TransporterStatus[vTi].LiftStationTarget := 0;
  TransporterStatus[vTi].SinkStationTarget := 0;
  TransporterStatus[vTi].XDriveTarget := vTargetX;
  TransporterStatus[vTi].XFinalTarget := vTargetX;

END_FOR;

STC_FC_TakeOut := TRUE;

END_FUNCTION

(* ---- STC_FC_TrackMoveTimes.st ---- *)
(* ===========================================================================================
 *  STC_FC_TrackMoveTimes — Record phase transition timestamps
 *
 *  Company : Galvatek part of the John Cockerill Group
 *  Author  : Jarmo Piipponen
 *  Created : 25.03.2026
 *
 * -------------------------------------------------------------------------------------------
 *  Called from SIM code at each transporter phase change.
 *  Uses Time100ms (0.1s ticks). On 4→0 completion,
 *  calculates net durations and updates Move[] with
 *  weighted average: new = (old * 4 + measured) / 5.
 *
 *  ------------------------------------------------------------------------------------------
 *
 *  Changes:
 *
 *
 *
 *)

FUNCTION STC_FC_TrackMoveTimes : BOOL

(* Introduction of Variables ----------------------------------------------------------------*)

VAR_INPUT
  iTrans                   : INT;   (* transporter index 1..MAX_TRANSPORTERS *)
  iPrev                    : INT;   (* previous phase *)
  iNew                     : INT;   (* new phase *)
END_VAR

VAR_EXTERNAL CONSTANT
    MAX_TRANSPORTERS        : INT;
    MIN_STATION_INDEX        : INT;
    MAX_STATION_INDEX        : INT;
END_VAR

VAR_EXTERNAL
  TransporterStatus             : ARRAY[1..MAX_TRANSPORTERS] OF UDT_TransporterStatusType;
  Stations                 : ARRAY[MIN_STATION_INDEX..MAX_STATION_INDEX] OF UDT_StationType;
  Transporters                     : ARRAY[0..MAX_TRANSPORTERS] OF UDT_TransporterType;
  Move                    : ARRAY[1..MAX_TRANSPORTERS] OF UDT_JC_MoveTimesType;
  ActualMove             : ARRAY[1..MAX_TRANSPORTERS] OF UDT_JC_ActualMoveTimeType;
  TimeS                  : LINT;
  Time100ms              : LINT;
END_VAR

VAR
  vT                         : INT;
  vLiftStn                  : INT;
  vSinkStn                  : INT;
  vStartStn                 : INT;
  vLi                        : INT;   (* lift station index = stn - 100 *)
  vSi                        : INT;   (* sink station index = stn - 100 *)
  vStI                      : INT;   (* start station index = stn - 100 *)
  vRawLift                  : INT;   (* measured lift duration in 0.1s ticks *)
  vRawSink                  : INT;   (* measured sink duration in 0.1s ticks *)
  vRawTrav1                 : INT;   (* measured travel start→lift in 0.1s ticks *)
  vRawTrav2                 : INT;   (* measured travel lift→sink in 0.1s ticks *)
  vDripX10                  : INT;   (* DrippingTime in 0.1s ticks from lift station *)
  vTrayX10                  : INT;   (* DripTrayDelay in 0.1s ticks from transporter config *)
  vDevX10                   : INT;   (* DeviceDelay in 0.1s ticks from sink station *)
END_VAR

vT := iTrans;

(* Bounds check *)
IF vT < 1 OR vT > MAX_TRANSPORTERS THEN
    RETURN;
END_IF;

CASE iPrev OF
    0: (* 0→1 : siirto nostoasemalle alkaa *)
        IF iNew = 1 THEN
            ActualMove[vT].StartStation := TransporterStatus[vT].CurrentStation;
            ActualMove[vT].LiftStation  := TransporterStatus[vT].LiftStationTarget;
            ActualMove[vT].SinkStation  := TransporterStatus[vT].SinkStationTarget;
            ActualMove[vT].ts0 := Time100ms;
            ActualMove[vT].Invalidated := FALSE;
        END_IF;
    1: (* 1→2 : nosto alkaa *)
        IF iNew = 2 THEN
            ActualMove[vT].ts1 := Time100ms;
        END_IF;
    2: (* 2→3 : siirto laskuasemalle alkaa *)
        IF iNew = 3 THEN
            ActualMove[vT].ts2 := Time100ms;
        END_IF;
    3: (* 3→4 : lasku alkaa *)
        IF iNew = 4 THEN
            ActualMove[vT].ts3 := Time100ms;
        END_IF;
    4: (* 4→0 : handled after CASE — see below *)
END_CASE;

(* ── Invalidate on anomaly (checked at every phase transition) ── *)
IF iNew > 0 THEN
    (* Not in automatic mode: task interrupted *)
    IF TransporterStatus[vT].Status < 4 THEN
        ActualMove[vT].Invalidated := TRUE;
    END_IF;
    (* Transporter fault active *)
    IF TransporterStatus[vT].Fault THEN
        ActualMove[vT].Invalidated := TRUE;
    END_IF;
END_IF;

(* ── 4→0 completion: calculate and update Move ── *)
IF iPrev = 4 AND iNew = 0 THEN
    ActualMove[vT].ts4 := Time100ms;

    (* Only update if all timestamps are valid and transfer was normal *)
    IF ActualMove[vT].ts0 > 0
       AND ActualMove[vT].ts1 > 0
       AND ActualMove[vT].ts2 > 0
       AND ActualMove[vT].ts3 > 0
       AND NOT ActualMove[vT].Invalidated
    THEN
                vLiftStn  := ActualMove[vT].LiftStation;
                vSinkStn  := ActualMove[vT].SinkStation;
                vStartStn := ActualMove[vT].StartStation;
                vLi   := vLiftStn  - MIN_STATION_INDEX;
                vSi   := vSinkStn  - MIN_STATION_INDEX;
                vStI := vStartStn - MIN_STATION_INDEX;

                (* Mechanical delays in 0.1s ticks *)
                vDripX10 := Stations[vLiftStn].DrippingTime;
                vTrayX10 := Transporters[vT].DripTrayDelay;
                vDevX10  := Stations[vSinkStn].DeviceDelay;

                (* Raw durations are already in 0.1s ticks *)
                vRawTrav1 := LINT_TO_INT(ActualMove[vT].ts1 - ActualMove[vT].ts0);
                vRawTrav2 := LINT_TO_INT(ActualMove[vT].ts3 - ActualMove[vT].ts2);

                (* Net lift = (ts2-ts1) - DrippingTime - DripTrayDelay *)
                vRawLift := LINT_TO_INT(ActualMove[vT].ts2 - ActualMove[vT].ts1)
                            - vDripX10 - vTrayX10;

                (* Net sink = (ts4-ts3) - DripTrayDelay - DeviceDelay *)
                vRawSink := LINT_TO_INT(ActualMove[vT].ts4 - ActualMove[vT].ts3)
                            - vTrayX10 - vDevX10;

                (* Clamp to minimum 0 *)
  IF vRawLift < 0 THEN vRawLift := 0; END_IF;
  IF vRawSink < 0 THEN vRawSink := 0; END_IF;
  IF vRawTrav1 < 0 THEN vRawTrav1 := 0; END_IF;
  IF vRawTrav2 < 0 THEN vRawTrav2 := 0; END_IF;

                (* Bounds check indices *)
                IF vLi >= 1 AND vLi <= 30
                   AND vSi >= 1 AND vSi <= 30
                   AND vStI >= 1 AND vStI <= 30
                THEN
                    (* Weighted average: new = (old * 4 + measured) / 5 *)

                    (* Lift time at lift station *)
                    Move[vT].LiftTime[vLi] :=
                        (Move[vT].LiftTime[vLi] * 4 + vRawLift) / 5;

                    (* Sink time at sink station *)
                    Move[vT].SinkTime[vSi] :=
                        (Move[vT].SinkTime[vSi] * 4 + vRawSink) / 5;

                    (* Travel: lift → sink (both directions) — phase 3 is always exact station-to-station *)
                    Move[vT].Travel[vLi].ToTime[vSi] :=
                        (Move[vT].Travel[vLi].ToTime[vSi] * 4 + vRawTrav2) / 5;
                    Move[vT].Travel[vSi].ToTime[vLi] :=
                        (Move[vT].Travel[vSi].ToTime[vLi] * 4 + vRawTrav2) / 5;
                END_IF;
            END_IF;
END_IF;

STC_FC_TrackMoveTimes := TRUE;

END_FUNCTION

(* ---- STC_FC_UpdateUnitLocation.st ---- *)
(* ===========================================================================================
 *  STC_FC_UpdateUnitLocation — Update a unit's location
 *
 *  Company : Galvatek part of the John Cockerill Group
 *  Author  : Jarmo Piipponen
 *  Created : 25.03.2026
 *
 * -------------------------------------------------------------------------------------------
 *  Sets Unit[iUnit].location to the given new location.
 *  Updates StationOccupancy[].UnitId + ChangeTime for both old
 *  and new locations.
 *
 *  When moving to a station:
 *  - Advances batch CurStage if batch is IN_PROCESS
 *  - Updates batch min/max/cal times from treatment program
 *  - Clears unit target if iNttPrimary = 1
 *
 *  ------------------------------------------------------------------------------------------
 *
 *  Changes:
 *
 *
 *
 *)

FUNCTION STC_FC_UpdateUnitLocation : BOOL

(* Introduction of Variables ----------------------------------------------------------------*)

VAR_INPUT
  iUnit                    : INT;   (* unit number to update *)
  iLocation                : INT;   (* new location: <100 = transporter id, >=100 = station number *)
  iNttPrimary             : INT;   (* 1 = sink is NTT primary → clear target, 0 = don't clear *)
END_VAR

VAR_EXTERNAL CONSTANT
    MAX_UNITS               : INT;
    MAX_TRANSPORTERS        : INT;
    MAX_STEPS_PER_PROGRAM   : INT;
    MIN_STATION_INDEX        : INT;
    MAX_STATION_INDEX        : INT;
    IN_PROCESS              : INT;
    USED                    : INT;
    TO_NONE                 : INT;
END_VAR

VAR_EXTERNAL
  Unit                    : ARRAY[1..MAX_UNITS] OF UDT_JC_UnitType;
  Stations                 : ARRAY[MIN_STATION_INDEX..MAX_STATION_INDEX] OF UDT_StationType;
  StationOccupancy             : ARRAY[1..MAX_STATION_INDEX] OF UDT_JC_UnitAtStationType;
  Batch                   : ARRAY[1..MAX_UNITS] OF UDT_BatchType;
  TreatmentPrograms                 : ARRAY[1..MAX_UNITS] OF UDT_TreatmentProgramType;
  TransporterStatus             : ARRAY[1..MAX_TRANSPORTERS] OF UDT_TransporterStatusType;
  Move                    : ARRAY[1..MAX_TRANSPORTERS] OF UDT_JC_MoveTimesType;
  TimeS                  : LINT;
END_VAR

VAR
  vOldLoc                   : INT;
  vNewStg                   : INT;
END_VAR

IF (iUnit >= 1) AND (iUnit <= MAX_UNITS) THEN
  vOldLoc := Unit[iUnit].location;

  (* --- Clear unit_id from old location (unified: transporter or station) --- *)
  IF (vOldLoc >= 1) AND (vOldLoc <= MAX_STATION_INDEX) THEN
    StationOccupancy[vOldLoc].UnitId     := 0;
    StationOccupancy[vOldLoc].ChangeTime := TimeS;
  END_IF;

  (* --- Update unit location --- *)
  Unit[iUnit].location := iLocation;

  (* --- Set unit_id on new location (unified: transporter or station) --- *)
  IF (iLocation >= 1) AND (iLocation <= MAX_STATION_INDEX) THEN
    StationOccupancy[iLocation].UnitId     := iUnit;
    StationOccupancy[iLocation].ChangeTime := TimeS;

    (* Station-specific: batch stage advance only when landing on a station *)
    IF (iLocation >= MIN_STATION_INDEX) THEN

    (* Advance batch stage if unit is USED with an active batch *)
    IF (Unit[iUnit].Status = USED)  (* USED *)
       AND (Batch[iUnit].BatchCode <> 0)
       AND (Batch[iUnit].State = IN_PROCESS)
       AND (Batch[iUnit].CurStage < MAX_STEPS_PER_PROGRAM) THEN
      Batch[iUnit].CurStage := Batch[iUnit].CurStage + 1;

      (* Stamp arrival time on new station — used by CalcSchedule for elapsed calculation *)
      Batch[iUnit].StartTime := TimeS;

      (* Update batch treatment times from program for the new stage *)
      IF (TreatmentPrograms[iUnit].ProgramId = Batch[iUnit].ProgId)
         AND (TreatmentPrograms[iUnit].ProgramId > 0) THEN
        vNewStg := Batch[iUnit].CurStage;
        IF (vNewStg >= 1) AND (vNewStg <= MAX_STEPS_PER_PROGRAM) THEN
          Batch[iUnit].MinTime := TreatmentPrograms[iUnit].Steps[vNewStg].MinTime;
          Batch[iUnit].MaxTime := TreatmentPrograms[iUnit].Steps[vNewStg].MaxTime;
          Batch[iUnit].CalTime := TreatmentPrograms[iUnit].Steps[vNewStg].CalTime;
        END_IF;
      END_IF;
    END_IF;

    (* NOT_PROCESSED batch on station: clear times so UI shows no progress bar *)
    IF (Batch[iUnit].BatchCode <> 0)
       AND (Batch[iUnit].State <> IN_PROCESS) THEN
      Batch[iUnit].MinTime   := 0;
      Batch[iUnit].CalTime   := 0;
      Batch[iUnit].MaxTime   := 32000;  (* ~8.9 h cap, INT max safe *)
      Batch[iUnit].StartTime := TimeS;
    END_IF;

    (* Clear unit target ONLY when iNttPrimary = 1 (primary NTT destination).
       All other cases: keep target so NTT retries primary later. *)
    IF Unit[iUnit].Target <> TO_NONE AND iNttPrimary > 0 THEN
      Unit[iUnit].Target := TO_NONE;  (* primary reached → clear *)
    END_IF;

    END_IF; (* iLocation >= MIN_STATION_INDEX — station-specific block *)
  END_IF; (* iLocation valid *)
END_IF;

STC_FC_UpdateUnitLocation := TRUE;

END_FUNCTION

(* ---- STC_FindStation.st ---- *)
(* ============================================================
   STC_FindStation — Find a station by its number

   Company : Galvatek part of the John Cockerill Group
   Author  : Jarmo Piipponen
   Created : 25.03.2026
   ============================================================
   Direct lookup in g_station[] by station number.
   Returns x_mm (DINT); other fields via VAR_OUTPUT.
   ------------------------------------------------------------
   Changes:
   ============================================================ *)

FUNCTION STC_FindStation : DINT   (* returns x_mm *)
VAR_INPUT
  station_number : INT;
END_VAR
VAR_OUTPUT
  found           : BOOL;
  skind           : INT;
  device_delay_s  : REAL;
  dropping_time_s : REAL;
END_VAR
VAR_EXTERNAL CONSTANT
    MIN_StationIndex : INT;
    MAX_StationIndex : INT;
END_VAR
VAR_EXTERNAL
  g_station : ARRAY[MIN_StationIndex..MAX_StationIndex] OF UDT_StationType;
END_VAR
VAR
  stn_data : UDT_StationType;
END_VAR

  (* Direct lookup by station number — no loop needed *)
  IF (station_number >= MIN_StationIndex) AND (station_number <= MAX_StationIndex) THEN
    stn_data := g_station[station_number];
    IF stn_data.TankId <> 0 THEN
      found := TRUE;
      STC_FindStation := stn_data.XPosition;
      skind := stn_data.DryWet;
      device_delay_s := INT_TO_REAL(stn_data.DeviceDelay) / 10.0;
      dropping_time_s := INT_TO_REAL(stn_data.DrippingTime) / 10.0;
      RETURN;
    END_IF;
  END_IF;

  found := FALSE;
  STC_FindStation := 0;
  skind := 0;
  device_delay_s := 0.0;
  dropping_time_s := 0.0;

END_FUNCTION

(* ---- STC_FindStationOffset.st ---- *)
(* ===========================================================================================
 *  STC_FindStationOffset — Find a station N steps away in a given direction
 *
 *  Company : Galvatek part of the John Cockerill Group
 *  Author  : Jarmo Piipponen / AI-assisted
 *  Created : 01.04.2026
 *
 * -------------------------------------------------------------------------------------------
 *  Starting from i_from_stn, walk i_dir direction (+1=right, -1=left) counting
 *  stations that belong to the transporter's task area.  Return the station number
 *  once i_min_steps stations have been passed, or 0 if not enough stations exist
 *  within the transporter's drive limits.
 *
 *  Only stations with TankId <> 0 are counted as real steps.
 *  The search is bounded by g_cfg[i_trans].DrivePosMin / DrivePosMax.
 *
 *  ------------------------------------------------------------------------------------------
 *
 *  Changes:
 *
 *
 *
 *)

FUNCTION STC_FindStationOffset : INT   (* returns station number or 0 *)

(* Introduction of Variables ----------------------------------------------------------------*)

VAR_INPUT
    i_trans     : INT;   (* transporter index — for drive limits and task area *)
    i_from_stn  : INT;   (* starting station *)
    i_dir       : INT;   (* +1 = right (increasing X), -1 = left (decreasing X) *)
    i_min_steps : INT;   (* minimum number of station steps to travel *)
END_VAR

VAR_EXTERNAL CONSTANT
    MIN_StationIndex  : INT;
    MAX_StationIndex  : INT;
    MAX_Transporters  : INT;
END_VAR

VAR_EXTERNAL
    g_station : ARRAY[MIN_StationIndex..MAX_StationIndex] OF UDT_StationType;
    g_cfg     : ARRAY[1..MAX_Transporters] OF UDT_TransporterType;
END_VAR

VAR
    from_x      : DINT;
    stn         : INT;
    steps       : INT;
    x           : DINT;
    drive_min   : DINT;
    drive_max   : DINT;
    in_area     : BOOL;
    ta          : INT;
END_VAR

(* Implementation ---------------------------------------------------------------------------*)

STC_FindStationOffset := 0;

(* Guard inputs *)
IF i_trans < 1 OR i_trans > MAX_Transporters THEN RETURN; END_IF;
IF i_from_stn < MIN_StationIndex OR i_from_stn > MAX_StationIndex THEN RETURN; END_IF;
IF i_dir <> 1 AND i_dir <> -1 THEN RETURN; END_IF;
IF i_min_steps < 1 THEN RETURN; END_IF;

from_x    := g_station[i_from_stn].XPosition;
drive_min := g_cfg[i_trans].DrivePosMin;
drive_max := g_cfg[i_trans].DrivePosMax;
steps     := 0;

(* Walk stations in the given direction.
   We scan the entire station range and check X-position relative to from_x
   in the chosen direction.  A simple linear scan is fast enough for ≤30 stations. *)

IF i_dir = 1 THEN
    (* Scan right: find stations with X > from_x, in ascending X order.
       Since station indices may not be in X-order, we do repeated nearest-next scans. *)
    FOR stn := MIN_StationIndex TO MAX_StationIndex DO
        (* skip dummy stations *)
        IF g_station[stn].TankId = 0 THEN CONTINUE; END_IF;

        x := g_station[stn].XPosition;
        IF x <= from_x THEN CONTINUE; END_IF;
        IF x > drive_max THEN CONTINUE; END_IF;

        (* Check task area membership *)
        in_area := FALSE;
        FOR ta := 1 TO 3 DO
            IF g_cfg[i_trans].TaskArea[ta].MinLift <> 0 THEN
                IF stn >= g_cfg[i_trans].TaskArea[ta].MinLift
                   AND stn <= g_cfg[i_trans].TaskArea[ta].MaxLift THEN
                    in_area := TRUE;
                END_IF;
                IF stn >= g_cfg[i_trans].TaskArea[ta].MinSink
                   AND stn <= g_cfg[i_trans].TaskArea[ta].MaxSink THEN
                    in_area := TRUE;
                END_IF;
            END_IF;
        END_FOR;
        IF NOT in_area THEN CONTINUE; END_IF;

        steps := steps + 1;
        IF steps >= i_min_steps THEN
            STC_FindStationOffset := stn;
            RETURN;
        END_IF;
    END_FOR;

ELSE  (* i_dir = -1 *)
    (* Scan left: find stations with X < from_x, in descending X order.
       Walk station indices from high to low — works when indices correlate with X. *)
    FOR stn := MAX_StationIndex TO MIN_StationIndex BY -1 DO
        IF g_station[stn].TankId = 0 THEN CONTINUE; END_IF;

        x := g_station[stn].XPosition;
        IF x >= from_x THEN CONTINUE; END_IF;
        IF x < drive_min THEN CONTINUE; END_IF;

        (* Check task area membership *)
        in_area := FALSE;
        FOR ta := 1 TO 3 DO
            IF g_cfg[i_trans].TaskArea[ta].MinLift <> 0 THEN
                IF stn >= g_cfg[i_trans].TaskArea[ta].MinLift
                   AND stn <= g_cfg[i_trans].TaskArea[ta].MaxLift THEN
                    in_area := TRUE;
                END_IF;
                IF stn >= g_cfg[i_trans].TaskArea[ta].MinSink
                   AND stn <= g_cfg[i_trans].TaskArea[ta].MaxSink THEN
                    in_area := TRUE;
                END_IF;
            END_IF;
        END_FOR;
        IF NOT in_area THEN CONTINUE; END_IF;

        steps := steps + 1;
        IF steps >= i_min_steps THEN
            STC_FindStationOffset := stn;
            RETURN;
        END_IF;
    END_FOR;
END_IF;

(* Not enough stations found *)
STC_FindStationOffset := 0;

(* ---- STC_ManualTask.st ---- *)
(* ===========================================================================================
 *  STC_ManualTask — Execute manual transport tasks from gateway
 *
 *  Company : Galvatek part of the John Cockerill Group
 *  Author  : Jarmo Piipponen
 *  Created : 25.03.2026
 *
 * -------------------------------------------------------------------------------------------
 *  For each transporter, checks g_manual_task[ti].Valid.
 *  If the transporter is idle (Phase=0), validates stations,
 *  calculates transfer time, and inserts a task into the queue
 *  (same pattern as TSK_NoTreatment).
 *  Clears Valid after task is created, or on invalid input.
 *
 *  Called from TSK_FB_Scheduler phase 2200 (before NTT).
 *
 * ------------------------------------------------------------------------------------------
 *
 *  Changes:
 *
 *
 *
 *)

FUNCTION STC_ManualTask : BOOL

(* Introduction of Variables ----------------------------------------------------------------*)

VAR_INPUT
  i_time_s                  : LINT;
END_VAR

VAR_IN_OUT
  io_task                   : ARRAY[1..MAX_TRANSPORTERS] OF UDT_JC_TskQueueType;
END_VAR

VAR_EXTERNAL
  g_manual_task             : ARRAY[1..MAX_TRANSPORTERS] OF UDT_JC_ManualTaskType;
  g_transporter             : ARRAY[1..MAX_TRANSPORTERS] OF UDT_TransporterStatusType;
  g_move                    : ARRAY[1..MAX_TRANSPORTERS] OF UDT_JC_MoveTimesType;
  g_unit                    : ARRAY[1..MAX_UNITS] OF UDT_JC_UnitType;
  Stations                  : ARRAY[MIN_STATION_INDEX..MAX_STATION_INDEX] OF UDT_StationType;
  Transporters              : ARRAY[0..MAX_TRANSPORTERS] OF UDT_TransporterType;
END_VAR

VAR_EXTERNAL CONSTANT
  MAX_TASK_QUEUE            : INT;
  MAX_UNITS                 : INT;
  USED                      : INT;
END_VAR

VAR
  ti                        : INT;
  ai                        : INT;
  sh                        : INT;
  lift                      : INT;
  sink                      : INT;
  covers                    : BOOL;
  trans_pos                 : INT;
  tmp_move                  : UDT_JC_MoveTimesType;
  xfer_s                    : REAL;
  travel_to_lift_s          : REAL;
  task_start                : LINT;
  task_end                  : LINT;
END_VAR

STC_ManualTask := TRUE;

FOR ti := 1 TO MAX_TRANSPORTERS DO
  IF NOT g_manual_task[ti].Valid THEN
    CONTINUE;
  END_IF;

  lift := g_manual_task[ti].LiftStation;
  sink := g_manual_task[ti].SinkStation;

  (* Validate station range *)
  IF lift < MIN_STATION_INDEX OR lift > MAX_STATION_INDEX
     OR sink < MIN_STATION_INDEX OR sink > MAX_STATION_INDEX
     OR lift = sink THEN
    g_manual_task[ti].Valid := FALSE;
    CONTINUE;
  END_IF;

  (* Transporter must be active and idle *)
  (* Transporter must be active and idle or in move-away *)
  IF NOT g_transporter[ti].IsActive THEN
    CONTINUE;
  END_IF;
  IF g_transporter[ti].Phase <> 0
     AND NOT (g_transporter[ti].Phase = 1 AND g_transporter[ti].Status = 3) THEN
    CONTINUE;  (* keep Valid — retry next cycle *)
  END_IF;

  (* Check lift station is within transporter TaskArea *)
  covers := FALSE;
  FOR ai := 1 TO 4 DO
    IF Transporters[ti].TaskArea[ai].MinLift > 0
       OR Transporters[ti].TaskArea[ai].MaxLift > 0 THEN
      IF lift >= Transporters[ti].TaskArea[ai].MinLift
         AND lift <= Transporters[ti].TaskArea[ai].MaxLift THEN
        covers := TRUE;
      END_IF;
    END_IF;
  END_FOR;

  IF NOT covers THEN
    g_manual_task[ti].Valid := FALSE;
    CONTINUE;
  END_IF;

  (* Calculate transfer time *)
  tmp_move := g_move[ti];
  xfer_s := STC_CalcTransferTime(
    i_from_stn            := lift,
    i_to_stn              := sink,
    i_move                := tmp_move,
    i_from_dropping_x10   := Stations[lift].DrippingTime,
    i_to_device_delay_x10 := Stations[sink].DeviceDelay,
    i_drip_tray_delay_x10 := Transporters[ti].DripTrayDelay);

  (* Calculate travel-to-lift: time for transporter to reach lift station *)
  travel_to_lift_s := 0.0;
  trans_pos := g_transporter[ti].CurrentStation;
  IF trans_pos > 0 AND trans_pos <> lift THEN
    travel_to_lift_s := STC_CalcHorizontalTravel(
      i_from_stn := trans_pos,
      i_to_stn   := lift,
      i_move     := tmp_move);
  END_IF;

  task_start := i_time_s + REAL_TO_LINT(travel_to_lift_s);
  task_end   := task_start + REAL_TO_LINT(xfer_s);

  (* Check sink station is free — no unit occupying it *)
  covers := TRUE;  (* reuse variable as sink_free flag *)
  FOR sh := 1 TO MAX_UNITS DO
    IF g_unit[sh].location = sink AND g_unit[sh].Status = USED THEN
      covers := FALSE;
    END_IF;
  END_FOR;
  IF NOT covers THEN
    g_manual_task[ti].Valid := FALSE;
    CONTINUE;
  END_IF;

  (* Insert task at queue position 1 *)
  IF io_task[ti].Count < MAX_TASK_QUEUE THEN
    FOR sh := io_task[ti].Count TO 1 BY -1 DO
      io_task[ti].Queue[sh + 1] := io_task[ti].Queue[sh];
    END_FOR;
    io_task[ti].Queue[1].Unit              := 0;
    io_task[ti].Queue[1].Stage             := 0;
    io_task[ti].Queue[1].LiftStationTarget := lift;
    io_task[ti].Queue[1].SinkStationTarget := sink;
    io_task[ti].Queue[1].StartTime         := task_start;
    io_task[ti].Queue[1].FinishTime        := task_end;
    io_task[ti].Queue[1].CalcTime          := 0;
    io_task[ti].Queue[1].MinTime           := 0;
    io_task[ti].Queue[1].MaxTime           := 0;
    io_task[ti].Queue[1].NttPrimary        := 0;
    io_task[ti].Count := io_task[ti].Count + 1;
  END_IF;

  g_manual_task[ti].Valid := FALSE;
END_FOR;

END_FUNCTION

(* ---- STC_MoveAway.st ---- *)
(* ===========================================================================================
 *  STC_MoveAway — Evaluate and trigger idle move-away for transporters
 *
 *  Company : Galvatek part of the John Cockerill Group
 *  Author  : Jarmo Piipponen / AI-assisted
 *  Created : 01.04.2026
 *
 * -------------------------------------------------------------------------------------------
 *  Called once per scheduler cycle (phase 2202).
 *  For each idle transporter (Phase=0, Status=3) sitting on a MoveAway station,
 *  checks if idle time exceeds the station's MoveAway threshold.
 *  If so, calculates a safe target station and initiates move-away by setting
 *  Phase:=1, Status:=3, LiftStationTarget:=dest_stn.
 *
 *  60-second rule: If the transporter's next queued task starts on the SAME station
 *  and begins within MOVE_AWAY_MIN_WAIT_S seconds, move-away is suppressed.
 *
 *  Direction fallback: If no station is found in the preferred direction, tries
 *  the opposite direction before giving up.
 *
 *  ------------------------------------------------------------------------------------------
 *
 *  Changes:
 *
 *
 *
 *)

FUNCTION STC_MoveAway : BOOL

(* Introduction of Variables ----------------------------------------------------------------*)

VAR_INPUT
    i_time_s : LINT;   (* current unix time in seconds *)
END_VAR

VAR_EXTERNAL CONSTANT
    MIN_StationIndex     : INT;
    MAX_StationIndex     : INT;
    MAX_Transporters     : INT;
    MOVE_AWAY_MIN_WAIT_S : LINT;
END_VAR

VAR_EXTERNAL
    g_transporter : ARRAY[1..MAX_Transporters] OF UDT_TransporterStatusType;
    g_station     : ARRAY[MIN_StationIndex..MAX_StationIndex] OF UDT_StationType;
    g_cfg         : ARRAY[1..MAX_Transporters] OF UDT_TransporterType;
    g_task        : ARRAY[1..MAX_Transporters] OF UDT_JC_TskQueueType;
    g_sim_trans   : ARRAY[1..MAX_Transporters] OF UDT_JC_SimTransporterType;
END_VAR

VAR
    ti            : INT;    (* transporter index *)
    stn           : INT;    (* current station *)
    move_away_s   : INT;    (* station's move-away threshold *)
    idle_time     : LINT;   (* seconds since idle start *)
    current_x     : DINT;   (* current X position *)
    next_lift_x   : DINT;   (* next task lift station X *)
    area_center   : DINT;   (* midpoint of drive area *)
    dir           : INT;    (* +1 = right, -1 = left *)
    dest_stn      : INT;    (* target station *)
    next_stn      : INT;    (* chain-search temp *)
    next_task_stn : INT;    (* next task start station *)
    time_to_start : LINT;   (* seconds until next task *)
END_VAR

(* Implementation ---------------------------------------------------------------------------*)

STC_MoveAway := TRUE;

FOR ti := 1 TO MAX_Transporters DO

    (* Only idle transporters in auto mode *)
    IF g_transporter[ti].Phase <> 0 THEN CONTINUE; END_IF;
    IF g_transporter[ti].Status <> 3 THEN CONTINUE; END_IF;
    IF NOT g_transporter[ti].IsActive THEN CONTINUE; END_IF;

    stn := g_transporter[ti].CurrentStation;
    IF stn < MIN_StationIndex OR stn > MAX_StationIndex THEN CONTINUE; END_IF;

    move_away_s := g_station[stn].MoveAway;
    IF move_away_s = 0 THEN CONTINUE; END_IF;

    (* Calculate idle time: seconds since last task completed *)
    idle_time := i_time_s - g_sim_trans[ti].IdleStartTime;
    IF idle_time < DINT_TO_LINT(INT_TO_DINT(move_away_s)) THEN CONTINUE; END_IF;

    (* 60-second rule: don't move away if next task starts on same station soon *)
    IF g_task[ti].Count > 0 THEN
        next_task_stn := g_task[ti].Queue[1].LiftStationTarget;
        IF next_task_stn = stn THEN
            time_to_start := g_task[ti].Queue[1].StartTime - i_time_s;
            IF time_to_start >= 0 AND time_to_start < MOVE_AWAY_MIN_WAIT_S THEN
                CONTINUE;
            END_IF;
        END_IF;
    END_IF;

    (* Idle time exceeded — calculate target *)
    current_x := g_transporter[ti].XPosition;

    (* Direction: toward next task, or toward area center *)
    IF g_task[ti].Count > 0 THEN
        next_lift_x := g_station[ g_task[ti].Queue[1].LiftStationTarget ].XPosition;
        IF next_lift_x > current_x THEN
            dir := 1;
        ELSE
            dir := -1;
        END_IF;
    ELSE
        area_center := (g_cfg[ti].DrivePosMin + g_cfg[ti].DrivePosMax) / 2;
        IF area_center > current_x THEN
            dir := 1;
        ELSE
            dir := -1;
        END_IF;
    END_IF;

    (* Find station at least 2 steps away *)
    dest_stn := STC_FindStationOffset(
        i_trans     := ti,
        i_from_stn  := stn,
        i_dir       := dir,
        i_min_steps := 2
    );

    (* Direction fallback: try opposite if first attempt failed *)
    IF dest_stn = 0 THEN
        dir := -dir;
        dest_stn := STC_FindStationOffset(
            i_trans     := ti,
            i_from_stn  := stn,
            i_dir       := dir,
            i_min_steps := 2
        );
        IF dest_stn = 0 THEN CONTINUE; END_IF;
    END_IF;

    (* Chain: skip consecutive MoveAway stations *)
    WHILE (dest_stn >= MIN_StationIndex) AND (dest_stn <= MAX_StationIndex)
          AND (g_station[dest_stn].MoveAway > 0) DO
        next_stn := STC_FindStationOffset(
            i_trans     := ti,
            i_from_stn  := dest_stn,
            i_dir       := dir,
            i_min_steps := 1
        );

        IF (next_stn = 0) OR (next_stn = dest_stn) THEN
            dest_stn := 0;
            EXIT;
        END_IF;

        dest_stn := next_stn;
    END_WHILE;

    IF dest_stn = 0 THEN CONTINUE; END_IF;

    (* Initiate move-away: Phase 1 + Status 3 = idle move *)
    g_transporter[ti].Phase := 1;
    (* Status stays 3 — auto idle *)
    g_transporter[ti].LiftStationTarget := dest_stn;
    g_transporter[ti].XDriveTarget := g_station[dest_stn].XPosition;
    g_transporter[ti].XFinalTarget := g_station[dest_stn].XPosition;

END_FOR;

(* ---- STC_NoTreatmentStates.st ---- *)
(* ===========================================================================================
 *  STC_NoTreatmentStates — Non-treatment target state management
 *
 *  Company : Galvatek part of the John Cockerill Group
 *  Author  : Jarmo Piipponen
 *  Created : 25.03.2026
 *
 * -------------------------------------------------------------------------------------------
 *  Manages non-treatment target states for all units.
 *
 *  Structure:
 *  Pass 0 — SNAPSHOT: read unit/batch/station state into snap[]
 *  Section 1 — PROCESSED: mark last-stage units as PROCESSED
 *  Section 2 — TO_AVOID: clear occupied next-stage stations
 *  Section 3 — TO_LOADING: route one empty unit to loading
 *
 *  ------------------------------------------------------------------------------------------
 *
 *  Changes:
 *
 *
 *
 *)

FUNCTION STC_NoTreatmentStates : BOOL

(* Introduction of Variables ----------------------------------------------------------------*)

VAR_EXTERNAL CONSTANT
    MAX_UNITS               : INT;
    MAX_STEPS_PER_PROGRAM   : INT;
    MAX_STATIONS_PER_STEP   : INT;
    MIN_STATION_INDEX        : INT;
    MAX_STATION_INDEX        : INT;
    IN_PROCESS              : INT;
    PROCESSED               : INT;
    NOT_USED                : INT;
    TO_NONE                 : INT;
    TO_UNLOAD               : INT;
    TO_AVOID                : INT;
    TO_LOADING              : INT;
    USED                    : INT;
    OP_BUFFER               : INT;
    OP_BUFFER_PROCESSED     : INT;
    OP_LOADING              : INT;
    OP_LOADING_UNLOADING    : INT;
END_VAR

VAR_EXTERNAL
  g_unit                    : ARRAY[1..MAX_UNITS] OF UDT_JC_UnitType;
  g_batch                   : ARRAY[1..MAX_UNITS] OF UDT_BatchType;
  TreatmentPrograms                 : ARRAY[1..MAX_UNITS] OF UDT_TreatmentProgramType;
  Stations                 : ARRAY[MIN_STATION_INDEX..MAX_STATION_INDEX] OF UDT_StationType;
  g_station_occupancy             : ARRAY[1..MAX_STATION_INDEX] OF UDT_JC_UnitAtStationType;
  g_time_s                  : LINT;
  g_production_queue        : INT;
  g_event_pending           : UDT_JC_EventMsgType;
  g_event_pending_valid     : BOOL;
END_VAR

VAR
  (* Snapshot *)
  snap                      : ARRAY[1..MAX_UNITS] OF UDT_JC_UnitSnapType;
  u                         : INT;        (* unit loop index *)
  has_loading               : BOOL;       (* any unit already has TO_LOADING *)
  (* Section 1+2 *)
  p                         : INT;        (* parallel station loop *)
  next_stn                  : INT;        (* next stage station *)
  occ_uid                   : INT;        (* unit_id at an occupied station *)
  free_found                : BOOL;       (* any next-stage station is free *)
  avoid_uid                 : INT;        (* unit to mark TO_AVOID *)
  (* Section 3 *)
  load_free                 : BOOL;       (* a loading station is free *)
  load_uid                  : INT;        (* best candidate for TO_LOADING *)
  load_in_buf               : BOOL;       (* current candidate is in buffer *)
  stk                       : INT;        (* station loop *)
  op                        : INT;        (* station operation code *)
END_VAR

  (* ════════════════════════════════════════════════════════════
     Pass 0 — SNAPSHOT: collect per-unit state in one pass
     ════════════════════════════════════════════════════════════ *)
  has_loading := FALSE;

  FOR u := 1 TO MAX_UNITS DO
    snap[u].IsActive := g_unit[u].Status <> NOT_USED;
    IF NOT snap[u].IsActive THEN
      CONTINUE;
    END_IF;

    snap[u].Location       := g_unit[u].location;
    snap[u].Target       := g_unit[u].Target;
    snap[u].HasBatch := g_batch[u].BatchCode <> 0;
    snap[u].BatchState    := g_batch[u].State;
    snap[u].CurStage := g_batch[u].CurStage;

    snap[u].OnStation := snap[u].Location >= MIN_STATION_INDEX
                          AND snap[u].Location <= MAX_STATION_INDEX;
    IF snap[u].OnStation THEN
      snap[u].LocationOp    := Stations[snap[u].Location].StationType;
      snap[u].InBuffer := snap[u].LocationOp >= OP_BUFFER AND snap[u].LocationOp <= OP_BUFFER_PROCESSED;
      IF g_station_occupancy[snap[u].Location].ChangeTime > 0 THEN
        snap[u].Elapsed := g_time_s - g_station_occupancy[snap[u].Location].ChangeTime;
      ELSE
        snap[u].Elapsed := 0;
      END_IF;
      IF snap[u].CurStage >= 1 THEN
        snap[u].CalTime := TreatmentPrograms[u].Steps[snap[u].CurStage].CalTime;
      ELSE
        snap[u].CalTime := 0;
      END_IF;
    ELSE
      snap[u].LocationOp    := 0;
      snap[u].InBuffer := FALSE;
      snap[u].Elapsed   := 0;
      snap[u].CalTime       := 0;
    END_IF;

    IF snap[u].Target = TO_LOADING THEN
      has_loading := TRUE;
    END_IF;
  END_FOR;

  (* ════════════════════════════════════════════════════════════
     Section 1 — PROCESSED: mark batch done at last treatment stage
     ════════════════════════════════════════════════════════════ *)
  FOR u := 1 TO MAX_UNITS DO
    IF NOT snap[u].IsActive OR NOT snap[u].HasBatch THEN
      CONTINUE;
    END_IF;
    IF snap[u].BatchState <> IN_PROCESS OR NOT snap[u].OnStation THEN
      CONTINUE;
    END_IF;
    IF snap[u].CurStage >= 1 AND snap[u].CurStage < MAX_STEPS_PER_PROGRAM THEN
      IF snap[u].CurStage >= TreatmentPrograms[u].StepCount THEN
        IF snap[u].Elapsed > 0 AND snap[u].Elapsed >= DINT_TO_LINT(snap[u].CalTime) THEN
          g_batch[u].State := PROCESSED;
          snap[u].BatchState   := PROCESSED;  (* update snapshot *)

          (* ── Emit BATCH_COMPLETED event (msg_type=5) ── *)
          IF NOT g_event_pending_valid THEN
            g_event_pending.MsgType := 5;
            g_event_pending.TsHi := LINT_TO_UINT(g_time_s / LINT#65536);
            g_event_pending.TsLo := LINT_TO_UINT(g_time_s MOD LINT#65536);
            g_event_pending.Payload[1]  := u;                                  (* unit_id *)
            g_event_pending.Payload[2]  := g_batch[u].BatchCode;               (* batch_code *)
            g_event_pending.Payload[3]  := TreatmentPrograms[u].StepCount;             (* stage_count *)
            g_event_pending.Payload[4]  := snap[u].Location;                   (* final_station *)
            g_event_pending.Payload[5]  := 0;
            g_event_pending.Payload[6]  := 0;
            g_event_pending.Payload[7]  := 0;
            g_event_pending.Payload[8]  := 0;
            g_event_pending.Payload[9]  := 0;
            g_event_pending.Payload[10] := 0;
            g_event_pending.Payload[11] := 0;
            g_event_pending.Payload[12] := 0;
            g_event_pending_valid := TRUE;
          END_IF;

          (* Route to unloading station *)
          IF snap[u].Target = TO_NONE THEN
            g_unit[u].Target := TO_UNLOAD;
            snap[u].Target   := TO_UNLOAD;
          END_IF;
        END_IF;
      END_IF;
    END_IF;
  END_FOR;

  (* ════════════════════════════════════════════════════════════
     Section 2 — TO_AVOID: clear the way to next treatment station
     ════════════════════════════════════════════════════════════ *)
  FOR u := 1 TO MAX_UNITS DO
    IF NOT snap[u].IsActive OR NOT snap[u].HasBatch THEN
      CONTINUE;
    END_IF;
    IF snap[u].BatchState <> IN_PROCESS THEN
      CONTINUE;
    END_IF;
    IF snap[u].CurStage < 1 OR snap[u].CurStage >= MAX_STEPS_PER_PROGRAM THEN
      CONTINUE;
    END_IF;
    IF snap[u].CurStage >= TreatmentPrograms[u].StepCount THEN
      CONTINUE;  (* no next stage *)
    END_IF;

    (* — Pass 1: any next-stage station free or being cleared? — *)
    free_found := FALSE;
    avoid_uid  := 0;
    FOR p := 0 TO MAX_STATIONS_PER_STEP - 1 DO
      next_stn := TreatmentPrograms[u].Steps[snap[u].CurStage + 1].Stations[p];
      IF next_stn = 0 THEN
        EXIT;
      END_IF;
      IF next_stn >= MIN_STATION_INDEX AND next_stn <= MAX_STATION_INDEX THEN
        IF g_station_occupancy[next_stn].UnitId = 0 THEN
          free_found := TRUE;
          EXIT;
        END_IF;
        occ_uid := g_station_occupancy[next_stn].UnitId;
        IF occ_uid >= 1 AND occ_uid <= MAX_UNITS THEN
          IF snap[occ_uid].Target = TO_AVOID THEN
            free_found := TRUE;
            EXIT;
          END_IF;
        END_IF;
      END_IF;
    END_FOR;

    (* — Pass 2: all occupied → mark ONE movable unit TO_AVOID — *)
    IF NOT free_found THEN
      FOR p := 0 TO MAX_STATIONS_PER_STEP - 1 DO
        next_stn := TreatmentPrograms[u].Steps[snap[u].CurStage + 1].Stations[p];
        IF next_stn = 0 THEN
          EXIT;
        END_IF;
        IF next_stn >= MIN_STATION_INDEX AND next_stn <= MAX_STATION_INDEX THEN
          occ_uid := g_station_occupancy[next_stn].UnitId;
          IF occ_uid >= 1 AND occ_uid <= MAX_UNITS THEN
            IF NOT snap[occ_uid].HasBatch AND snap[occ_uid].Target = TO_NONE THEN
              avoid_uid := occ_uid;
              EXIT;
            END_IF;
          END_IF;
        END_IF;
      END_FOR;

      IF avoid_uid >= 1 THEN
        g_unit[avoid_uid].Target := TO_AVOID;
        snap[avoid_uid].Target     := TO_AVOID;  (* update snapshot *)
      END_IF;
    END_IF;
  END_FOR;

  (* ════════════════════════════════════════════════════════════
     Section 3 — TO_LOADING: route one empty unit to loading station
     ════════════════════════════════════════════════════════════ *)
  IF g_production_queue = 1 AND NOT has_loading THEN

    (* Check if any loading station is free *)
    load_free := FALSE;
    FOR stk := MIN_STATION_INDEX TO MAX_STATION_INDEX DO
      op := Stations[stk].StationType;
      IF (op = OP_LOADING OR op = OP_LOADING_UNLOADING)
         AND g_station_occupancy[stk].UnitId = 0 THEN
        load_free := TRUE;
        EXIT;
      END_IF;
    END_FOR;

    IF load_free THEN
      load_uid    := 0;
      load_in_buf := FALSE;
      FOR u := 1 TO MAX_UNITS DO
        IF snap[u].IsActive AND NOT snap[u].HasBatch
           AND snap[u].Target = TO_NONE AND snap[u].OnStation THEN
          IF snap[u].InBuffer THEN
            IF load_uid = 0 THEN
              load_uid    := u;
              load_in_buf := TRUE;
            END_IF;
          ELSE
            IF load_uid = 0 OR load_in_buf THEN
              load_uid    := u;
              load_in_buf := FALSE;
            END_IF;
          END_IF;
        END_IF;
      END_FOR;

      IF load_uid >= 1 THEN
        g_unit[load_uid].Target := TO_LOADING;
      END_IF;
    END_IF; (* load_free *)

  END_IF; (* production_queue AND NOT has_loading *)

  STC_NoTreatmentStates := TRUE;

END_FUNCTION

(* ---- STC_ShiftSchedule.st ---- *)
(* ===========================================================================================
 *  STC_ShiftSchedule — Shift schedule + task times
 *
 *  Company : Galvatek part of the John Cockerill Group
 *  Author  : Jarmo Piipponen
 *  Created : 25.03.2026
 *
 * -------------------------------------------------------------------------------------------
 *  Propagates a time shift through one unit's schedule stages
 *  AND through all matching tasks.
 *
 *  Positive i_amount = DELAY (shift later),
 *  Negative i_amount = ADVANCE (shift earlier).
 *
 *  VAR_IN_OUT: io_schedule, io_task — caller passes live or
 *  workspace arrays.
 *
 *  ------------------------------------------------------------------------------------------
 *
 *  Changes:
 *
 *
 *
 *)

FUNCTION STC_ShiftSchedule : BOOL

(* Introduction of Variables ----------------------------------------------------------------*)

VAR_INPUT
  i_unit                    : INT;     (* unit index 1..10 *)
  i_from_stage              : INT;     (* propagate from this stage onward *)
  i_amount                  : REAL;    (* seconds to shift (+ = later, - = earlier) *)
END_VAR

VAR_IN_OUT  (* array sizes must match GVL_JC_Constants: 10=MAX_UNITS, 3=MAX_TRANSPORTERS *)
  io_schedule               : ARRAY[1..10] OF UDT_JC_TskScheduleType;
  io_task                   : ARRAY[1..3] OF UDT_JC_TskQueueType;
END_VAR

VAR_EXTERNAL CONSTANT
    MAX_TRANSPORTERS        : INT;
    MAX_UNITS               : INT;
END_VAR

VAR_EXTERNAL
  g_time_s                  : LINT;
END_VAR

VAR
  sc                        : INT;
  si                        : INT;
  qi                        : INT;
  ti                        : INT;
  duration                  : LINT;
END_VAR

STC_ShiftSchedule := TRUE;
IF i_unit < 1 OR i_unit > MAX_UNITS THEN RETURN; END_IF;
IF ABS(i_amount) < 0.001 THEN RETURN; END_IF;

(* -- Shift schedule stages entry/exit times -- *)
sc := io_schedule[i_unit].StageCount;
FOR si := 1 TO sc DO
  IF si >= 1 AND si <= 30
     AND io_schedule[i_unit].Stages[si].ProgramStage >= i_from_stage THEN
    io_schedule[i_unit].Stages[si].EntryTime :=
      io_schedule[i_unit].Stages[si].EntryTime + REAL_TO_LINT(i_amount);
    io_schedule[i_unit].Stages[si].ExitTime :=
      io_schedule[i_unit].Stages[si].ExitTime + REAL_TO_LINT(i_amount);
    (* GAP-3: Past-clamp -- don't let EntryTime go before now+1 *)
    IF i_amount < 0.0 AND io_schedule[i_unit].Stages[si].EntryTime < g_time_s + LINT#1 THEN
      io_schedule[i_unit].Stages[si].ExitTime := g_time_s + LINT#1
        + (io_schedule[i_unit].Stages[si].ExitTime - io_schedule[i_unit].Stages[si].EntryTime);
      io_schedule[i_unit].Stages[si].EntryTime := g_time_s + LINT#1;
    END_IF;
  END_IF;
END_FOR;

(* -- Shift matching tasks in all transporter queues -- *)
FOR ti := 1 TO MAX_TRANSPORTERS DO
  FOR qi := 1 TO io_task[ti].Count DO
    IF io_task[ti].Queue[qi].Unit = i_unit
       AND io_task[ti].Queue[qi].Stage >= i_from_stage THEN
      io_task[ti].Queue[qi].StartTime :=
        io_task[ti].Queue[qi].StartTime + REAL_TO_LINT(i_amount);
      io_task[ti].Queue[qi].FinishTime :=
        io_task[ti].Queue[qi].FinishTime + REAL_TO_LINT(i_amount);
      (* GAP-3: Past-clamp -- don't let StartTime go before now+1 *)
      IF i_amount < 0.0 AND io_task[ti].Queue[qi].StartTime < g_time_s + LINT#1 THEN
        duration := io_task[ti].Queue[qi].FinishTime - io_task[ti].Queue[qi].StartTime;
        io_task[ti].Queue[qi].StartTime := g_time_s + LINT#1;
        io_task[ti].Queue[qi].FinishTime := g_time_s + LINT#1 + duration;
      END_IF;
    END_IF;
  END_FOR;
END_FOR;

END_FUNCTION
